C09083=1072.858,202.514,-79.918,173.836,27.136,154.832
C09084=1072.852,202.266,-79.894,173.834,27.133,154.832
C09085=1072.846,202.016,-79.870,173.831,27.130,154.831
C09086=1072.840,201.767,-79.847,173.830,27.128,154.831
C09087=1072.835,201.519,-79.822,173.827,27.125,154.831
C09088=1072.828,201.270,-79.798,173.825,27.122,154.830
C09089=1072.823,201.021,-79.774,173.822,27.119,154.830
C09090=1072.817,200.772,-79.751,173.820,27.116,154.830
C09091=1072.811,200.524,-79.727,173.819,27.114,154.829
C09092=1072.805,200.275,-79.703,173.816,27.110,154.829
C09093=1072.800,200.026,-79.680,173.814,27.107,154.828
C09094=1072.794,199.777,-79.656,173.811,27.104,154.828
C09095=1072.788,199.529,-79.632,173.810,27.102,154.828
C09096=1072.783,199.279,-79.608,173.807,27.099,154.827
C09097=1072.777,199.031,-79.584,173.805,27.096,154.827
C09098=1072.771,198.783,-79.561,173.802,27.093,154.827
C09099=1072.766,198.533,-79.537,173.801,27.090,154.826
C09100=1072.759,198.284,-79.513,173.799,27.087,154.826
C09101=1072.754,198.035,-79.490,173.796,27.085,154.826
C09102=1072.748,197.787,-79.466,173.794,27.082,154.825
C09103=1072.743,197.538,-79.442,173.792,27.079,154.825
C09104=1072.737,197.289,-79.419,173.790,27.076,154.824
C09105=1072.730,197.040,-79.395,173.787,27.073,154.824
C09106=1072.725,196.791,-79.371,173.785,27.070,154.824
C09107=1072.719,196.543,-79.348,173.783,27.068,154.823
C09108=1072.714,196.294,-79.325,173.781,27.065,154.823
C09109=1072.708,196.045,-79.300,173.779,27.062,154.823
C09110=1072.702,195.797,-79.277,173.776,27.059,154.822
C09111=1072.697,195.547,-79.253,173.775,27.056,154.822
C09112=1072.691,195.298,-79.230,173.772,27.053,154.821
C09113=1072.685,195.050,-79.206,173.770,27.050,154.821
C09114=1072.680,194.801,-79.183,173.768,27.047,154.821
C09115=1072.674,194.552,-79.160,173.766,27.044,154.820
C09116=1072.668,194.304,-79.136,173.764,27.041,154.820
C09117=1072.663,194.054,-79.112,173.761,27.039,154.820
C09118=1072.657,193.806,-79.089,173.760,27.036,154.819
C09119=1072.651,193.556,-79.065,173.757,27.033,154.819
C09120=1072.646,193.307,-79.042,173.755,27.030,154.818
C09121=1072.640,193.059,-79.018,173.753,27.027,154.818
C09122=1072.635,192.810,-78.995,173.751,27.025,154.818
C09123=1072.629,192.562,-78.971,173.748,27.022,154.817
C09124=1072.623,192.313,-78.948,173.747,27.019,154.817
C09125=1072.618,192.064,-78.925,173.745,27.016,154.817
C09126=1072.612,191.815,-78.901,173.742,27.013,154.816
C09127=1072.606,191.533,-78.875,173.740,27.010,154.816
C09128=1072.599,191.252,-78.848,173.737,27.007,154.815
C09129=1072.593,190.970,-78.822,173.735,27.003,154.815
C09130=1072.587,190.689,-78.796,173.733,27.000,154.815
C09131=1072.581,190.441,-78.772,173.730,26.997,154.814
C09132=1072.575,190.192,-78.749,173.729,26.994,154.814
C09133=1072.570,189.943,-78.726,173.726,26.991,154.813
C09134=1072.565,189.694,-78.703,173.724,26.989,154.813
C09135=1072.559,189.445,-78.679,173.722,26.986,154.813
C09136=1072.553,189.196,-78.656,173.720,26.983,154.812
C09137=1072.548,188.947,-78.633,173.718,26.980,154.812
C09138=1072.542,188.698,-78.610,173.716,26.977,154.811
C09139=1072.537,188.449,-78.587,173.714,26.974,154.811
C09140=1072.531,188.201,-78.563,173.711,26.972,154.811
C09141=1072.526,187.952,-78.539,173.710,26.969,154.810
C09142=1072.520,187.703,-78.517,173.707,26.966,154.810
C09143=1072.514,187.454,-78.494,173.705,26.963,154.810
C09144=1072.508,187.205,-78.471,173.704,26.960,154.809
C09145=1072.503,186.956,-78.447,173.701,26.957,154.809
C09146=1072.498,186.707,-78.424,173.700,26.955,154.809
C09147=1072.492,186.458,-78.401,173.697,26.952,154.808
C09148=1072.486,186.209,-78.378,173.695,26.949,154.808
C09149=1072.481,185.961,-78.354,173.693,26.946,154.807
C09150=1072.475,185.712,-78.331,173.691,26.943,154.807
C09151=1072.469,185.463,-78.308,173.689,26.940,154.807
C09152=1072.464,185.215,-78.286,173.687,26.937,154.806
C09153=1072.459,184.966,-78.262,173.685,26.934,154.806
C09154=1072.454,184.717,-78.239,173.682,26.931,154.806
C09155=1072.448,184.468,-78.216,173.681,26.929,154.805
C09156=1072.441,184.219,-78.194,173.678,26.926,154.805
C09157=1072.436,183.970,-78.171,173.677,26.923,154.804
C09158=1072.430,183.721,-78.148,173.674,26.921,154.804
C09159=1072.424,183.472,-78.126,173.672,26.918,154.804
C09160=1072.419,183.223,-78.103,173.671,26.915,154.803
C09161=1072.413,182.974,-78.080,173.668,26.912,154.803
C09162=1072.407,182.725,-78.057,173.666,26.909,154.803
C09163=1072.401,182.477,-78.034,173.664,26.907,154.802
C09164=1072.395,182.228,-78.012,173.662,26.904,154.802
C09165=1072.389,181.979,-77.989,173.660,26.901,154.802
C09166=1072.384,181.730,-77.966,173.658,26.899,154.801
C09167=1072.377,181.481,-77.943,173.655,26.896,154.801
C09168=1072.372,181.232,-77.921,173.654,26.893,154.801
C09169=1072.366,180.983,-77.898,173.651,26.890,154.800
C09170=1072.360,180.734,-77.875,173.650,26.888,154.800
C09171=1072.355,180.485,-77.852,173.647,26.885,154.800
C09172=1072.348,180.237,-77.830,173.645,26.882,154.799
C09173=1072.343,179.987,-77.808,173.644,26.880,154.799
C09174=1072.337,179.738,-77.785,173.641,26.877,154.799
C09175=1072.331,179.489,-77.762,173.640,26.874,154.798
C09176=1072.325,179.240,-77.739,173.637,26.871,154.798
C09177=1072.319,178.992,-77.716,173.635,26.868,154.798
C09178=1072.314,178.743,-77.695,173.633,26.866,154.797
C09179=1072.308,178.494,-77.672,173.631,26.863,154.797
C09180=1072.303,178.245,-77.649,173.629,26.860,154.796
C09181=1072.296,177.996,-77.627,173.627,26.858,154.796
C09182=1072.291,177.747,-77.604,173.625,26.855,154.796
C09183=1072.285,177.498,-77.581,173.623,26.852,154.795
C09184=1072.280,177.249,-77.559,173.621,26.849,154.795
C09185=1072.273,177.000,-77.537,173.619,26.847,154.795
C09186=1072.268,176.752,-77.514,173.617,26.844,154.794
C09187=1072.263,176.502,-77.492,173.615,26.841,154.794
C09188=1072.257,176.253,-77.469,173.613,26.838,154.794
C09189=1072.250,176.005,-77.446,173.610,26.836,154.793
C09190=1072.245,175.755,-77.424,173.609,26.833,154.793
C09191=1072.239,175.475,-77.399,173.607,26.830,154.793
C09192=1072.233,175.192,-77.373,173.604,26.827,154.792
C09193=1072.226,174.910,-77.348,173.602,26.824,154.792
C09194=1072.219,174.629,-77.322,173.599,26.821,154.792
C09195=1072.213,174.379,-77.300,173.598,26.818,154.791
C09196=1072.208,174.131,-77.277,173.596,26.815,154.791
C09197=1072.202,173.882,-77.256,173.594,26.813,154.790
C09198=1072.196,173.633,-77.233,173.592,26.810,154.790
C09199=1072.191,173.383,-77.211,173.590,26.807,154.790
C09200=1072.185,173.135,-77.189,173.588,26.804,154.789
C09201=1072.180,172.886,-77.166,173.586,26.802,154.789
C09202=1072.174,172.637,-77.144,173.584,26.798,154.789
C09203=1072.168,172.388,-77.122,173.581,26.796,154.788
C09204=1072.163,172.140,-77.099,173.580,26.793,154.788
C09205=1072.157,171.890,-77.077,173.578,26.790,154.788
C09206=1072.151,171.641,-77.055,173.576,26.788,154.787
C09207=1072.145,171.392,-77.032,173.574,26.785,154.787
C09208=1072.140,171.143,-77.011,173.572,26.782,154.786
C09209=1072.134,170.895,-76.988,173.570,26.779,154.786
C09210=1072.129,170.645,-76.966,173.568,26.777,154.786
C09211=1072.123,170.397,-76.943,173.566,26.774,154.785
C09212=1072.117,170.148,-76.922,173.564,26.771,154.785
C09213=1072.112,169.898,-76.900,173.562,26.768,154.785
C09214=1072.107,169.650,-76.877,173.561,26.765,154.784
C09215=1072.101,169.401,-76.855,173.558,26.762,154.784
C09216=1072.095,169.152,-76.832,173.557,26.760,154.784
C09217=1072.089,168.902,-76.810,173.554,26.757,154.783
C09218=1072.084,168.654,-76.789,173.553,26.754,154.783
C09219=1072.078,168.405,-76.766,173.550,26.752,154.783
C09220=1072.073,168.156,-76.744,173.549,26.749,154.782
C09221=1072.067,167.907,-76.722,173.546,26.746,154.782
C09222=1072.062,167.657,-76.700,173.545,26.744,154.781
C09223=1072.056,167.410,-76.678,173.543,26.741,154.781
C09224=1072.050,167.160,-76.656,173.541,26.738,154.781
C09225=1072.045,166.910,-76.634,173.539,26.735,154.780
C09226=1072.039,166.663,-76.612,173.537,26.733,154.780
C09227=1072.034,166.413,-76.590,173.535,26.729,154.780
C09228=1072.028,166.165,-76.568,173.533,26.727,154.779
C09229=1072.023,165.915,-76.546,173.531,26.724,154.779
C09230=1072.017,165.666,-76.524,173.529,26.721,154.779
C09231=1072.011,165.418,-76.502,173.527,26.718,154.778
C09232=1072.006,165.168,-76.480,173.526,26.715,154.778
C09233=1072.000,164.920,-76.458,173.523,26.713,154.778
C09234=1071.995,164.670,-76.436,173.522,26.710,154.777
C09235=1071.990,164.421,-76.414,173.519,26.707,154.777
C09236=1071.984,164.173,-76.392,173.518,26.704,154.776
C09237=1071.978,163.923,-76.370,173.516,26.702,154.776
C09238=1071.973,163.675,-76.348,173.514,26.699,154.776
C09239=1071.967,163.425,-76.326,173.513,26.696,154.775
C09240=1071.962,163.177,-76.305,173.510,26.693,154.775
C09241=1071.956,162.927,-76.283,173.509,26.691,154.775
C09242=1071.951,162.679,-76.261,173.506,26.688,154.774
C09243=1071.945,162.429,-76.239,173.505,26.685,154.774
C09244=1071.940,162.180,-76.217,173.503,26.682,154.773
C09245=1071.934,161.931,-76.196,173.501,26.680,154.773
C09246=1071.929,161.683,-76.173,173.499,26.677,154.773
C09247=1071.923,161.434,-76.151,173.497,26.674,154.772
C09248=1071.918,161.185,-76.130,173.496,26.671,154.772
C09249=1071.912,160.936,-76.108,173.493,26.668,154.772
C09250=1071.906,160.687,-76.087,173.492,26.666,154.771
C09251=1071.900,160.438,-76.065,173.489,26.663,154.771
C09252=1071.895,160.188,-76.043,173.488,26.660,154.771
C09253=1071.889,159.940,-76.022,173.486,26.657,154.770
C09254=1071.883,159.690,-76.001,173.484,26.655,154.770
C09255=1071.877,159.409,-75.976,173.482,26.652,154.770
C09256=1071.871,159.126,-75.952,173.479,26.649,154.769
C09257=1071.864,158.844,-75.927,173.478,26.646,154.769
C09258=1071.858,158.561,-75.902,173.476,26.643,154.768
C09259=1071.852,158.313,-75.881,173.473,26.640,154.768
C09260=1071.846,158.064,-75.859,173.472,26.637,154.768
C09261=1071.840,157.815,-75.838,173.469,26.634,154.767
C09262=1071.834,157.566,-75.816,173.468,26.632,154.767
C09263=1071.830,157.316,-75.795,173.466,26.629,154.767
C09264=1071.824,157.067,-75.774,173.464,26.626,154.766
C09265=1071.818,156.819,-75.752,173.463,26.624,154.766
C09266=1071.812,156.569,-75.731,173.460,26.621,154.766
C09267=1071.806,156.321,-75.709,173.459,26.618,154.765
C09268=1071.801,156.071,-75.687,173.456,26.615,154.765
C09269=1071.796,155.822,-75.667,173.455,26.613,154.764
C09270=1071.789,155.573,-75.645,173.453,26.610,154.764
C09271=1071.784,155.325,-75.624,173.451,26.608,154.764
C09272=1071.778,155.075,-75.602,173.449,26.605,154.763
C09273=1071.772,154.827,-75.581,173.447,26.602,154.763
C09274=1071.766,154.577,-75.560,173.446,26.599,154.763
C09275=1071.761,154.329,-75.539,173.444,26.597,154.762
C09276=1071.755,154.079,-75.516,173.442,26.594,154.762
C09277=1071.750,153.831,-75.495,173.440,26.591,154.762
C09278=1071.745,153.581,-75.475,173.438,26.589,154.761
C09279=1071.738,153.332,-75.453,173.436,26.586,154.761
C09280=1071.733,153.084,-75.432,173.435,26.583,154.761
C09281=1071.727,152.834,-75.411,173.432,26.581,154.760
C09282=1071.721,152.585,-75.390,173.431,26.578,154.760
C09283=1071.715,152.336,-75.368,173.429,26.575,154.760
C09284=1071.710,152.087,-75.347,173.427,26.572,154.759
C09285=1071.704,151.838,-75.326,173.426,26.570,154.759
C09286=1071.698,151.589,-75.304,173.423,26.567,154.759
C09287=1071.693,151.340,-75.284,173.422,26.564,154.758
C09288=1071.687,151.091,-75.262,173.419,26.561,154.758
C09289=1071.681,150.843,-75.241,173.418,26.559,154.757
C09290=1071.675,150.593,-75.220,173.417,26.556,154.757
C09291=1071.670,150.344,-75.199,173.414,26.554,154.757
C09292=1071.665,150.095,-75.178,173.413,26.551,154.756
C09293=1071.658,149.846,-75.157,173.411,26.548,154.756
C09294=1071.653,149.597,-75.135,173.409,26.545,154.756
C09295=1071.647,149.348,-75.114,173.407,26.543,154.755
C09296=1071.641,149.099,-75.093,173.405,26.540,154.755
C09297=1071.636,148.850,-75.073,173.403,26.537,154.755
C09298=1071.630,148.601,-75.051,173.402,26.534,154.754
C09299=1071.625,148.352,-75.030,173.400,26.532,154.754
C09300=1071.619,148.102,-75.009,173.398,26.529,154.754
C09301=1071.613,147.853,-74.988,173.397,26.527,154.753
C09302=1071.608,147.605,-74.967,173.394,26.524,154.753
C09303=1071.602,147.355,-74.946,173.393,26.521,154.753
C09304=1071.596,147.107,-74.925,173.390,26.518,154.752
C09305=1071.590,146.858,-74.905,173.389,26.516,154.752
C09306=1071.584,146.608,-74.883,173.387,26.513,154.752
C09307=1071.579,146.359,-74.863,173.385,26.510,154.751
C09308=1071.573,146.109,-74.842,173.384,26.508,154.751
C09309=1071.567,145.861,-74.821,173.382,26.505,154.750
C09310=1071.562,145.612,-74.800,173.380,26.502,154.750
C09311=1071.555,145.363,-74.779,173.378,26.500,154.750
C09312=1071.550,145.114,-74.758,173.377,26.497,154.749
C09313=1071.545,144.865,-74.738,173.374,26.494,154.749
C09314=1071.539,144.615,-74.716,173.373,26.492,154.749
C09315=1071.533,144.367,-74.696,173.371,26.489,154.748
C09316=1071.527,144.118,-74.676,173.369,26.486,154.748
C09317=1071.521,143.868,-74.654,173.368,26.484,154.748
C09318=1071.516,143.619,-74.633,173.366,26.481,154.747
C09319=1071.509,143.337,-74.610,173.364,26.478,154.747
C09320=1071.503,143.054,-74.586,173.361,26.475,154.747
C09321=1071.496,142.772,-74.563,173.360,26.472,154.746
C09322=1071.490,142.489,-74.540,173.358,26.469,154.746
C09323=1071.484,142.241,-74.519,173.356,26.466,154.745
C09324=1071.479,141.991,-74.498,173.354,26.463,154.745
C09325=1071.473,141.742,-74.477,173.352,26.461,154.745
C09326=1071.467,141.494,-74.456,173.351,26.458,154.744
C09327=1071.461,141.244,-74.436,173.349,26.455,154.744
C09328=1071.456,140.995,-74.415,173.347,26.453,154.744
C09329=1071.451,140.746,-74.394,173.346,26.450,154.743
C09330=1071.444,140.498,-74.374,173.343,26.447,154.743
C09331=1071.438,140.248,-74.353,173.342,26.445,154.743
C09332=1071.433,139.999,-74.332,173.340,26.442,154.742
C09333=1071.427,139.750,-74.312,173.338,26.439,154.742
C09334=1071.422,139.501,-74.292,173.337,26.436,154.742
C09335=1071.416,139.251,-74.271,173.335,26.434,154.741
C09336=1071.410,139.003,-74.250,173.333,26.431,154.741
C09337=1071.405,138.754,-74.230,173.331,26.428,154.740
C09338=1071.399,138.504,-74.209,173.330,26.426,154.740
C09339=1071.393,138.255,-74.189,173.327,26.423,154.740
C09340=1071.387,138.006,-74.168,173.326,26.421,154.740
C09341=1071.381,137.757,-74.148,173.325,26.418,154.739
C09342=1071.376,137.508,-74.128,173.323,26.415,154.739
C09343=1071.370,137.258,-74.107,173.321,26.412,154.738
C09344=1071.364,137.010,-74.086,173.319,26.410,154.738
C09345=1071.359,136.761,-74.066,173.318,26.407,154.738
C09346=1071.353,136.512,-74.046,173.315,26.404,154.737
C09347=1071.348,136.263,-74.025,173.314,26.402,154.737
C09348=1071.341,136.013,-74.005,173.312,26.399,154.737
C09349=1071.336,135.764,-73.984,173.310,26.396,154.736
C09350=1071.330,135.515,-73.964,173.309,26.394,154.736
C09351=1071.324,135.266,-73.944,173.307,26.391,154.736
C09352=1071.318,135.017,-73.924,173.306,26.389,154.735
C09353=1071.313,134.768,-73.903,173.303,26.386,154.735
C09354=1071.307,134.519,-73.883,173.302,26.383,154.735
C09355=1071.301,134.270,-73.862,173.300,26.380,154.734
C09356=1071.295,134.021,-73.842,173.298,26.377,154.734
C09357=1071.290,133.772,-73.822,173.297,26.375,154.734
C09358=1071.285,133.523,-73.801,173.295,26.372,154.733
C09359=1071.278,133.273,-73.781,173.293,26.369,154.733
C09360=1071.273,133.024,-73.760,173.291,26.367,154.733
C09361=1071.267,132.775,-73.740,173.290,26.364,154.732
C09362=1071.262,132.525,-73.721,173.289,26.361,154.732
C09363=1071.256,132.277,-73.701,173.286,26.359,154.731
C09364=1071.251,132.027,-73.680,173.285,26.356,154.731
C09365=1071.245,131.779,-73.660,173.283,26.354,154.731
C09366=1071.238,131.529,-73.640,173.282,26.351,154.730
C09367=1071.232,131.280,-73.620,173.279,26.348,154.730
C09368=1071.227,131.031,-73.599,173.278,26.345,154.730
C09369=1071.221,130.782,-73.579,173.276,26.343,154.729
C09370=1071.215,130.533,-73.560,173.274,26.340,154.729
C09371=1071.209,130.283,-73.539,173.273,26.338,154.729
C09372=1071.203,130.034,-73.519,173.271,26.335,154.728
C09373=1071.197,129.785,-73.499,173.270,26.333,154.728
C09374=1071.191,129.537,-73.479,173.267,26.330,154.728
C09375=1071.186,129.287,-73.459,173.266,26.327,154.727
C09376=1071.180,129.038,-73.439,173.264,26.324,154.727
C09377=1071.174,128.789,-73.419,173.263,26.322,154.727
C09378=1071.168,128.540,-73.399,173.261,26.319,154.726
C09379=1071.163,128.291,-73.379,173.259,26.316,154.726
C09380=1071.157,128.041,-73.359,173.258,26.314,154.726
C09381=1071.151,127.792,-73.339,173.255,26.311,154.725
C09382=1071.145,127.544,-73.319,173.254,26.309,154.725
C09383=1071.138,127.261,-73.296,173.252,26.306,154.725
C09384=1071.132,126.978,-73.274,173.250,26.303,154.724
C09385=1071.126,126.695,-73.252,173.249,26.300,154.724
C09386=1071.118,126.413,-73.229,173.246,26.297,154.723
C09387=1071.113,126.163,-73.209,173.245,26.294,154.723
C09388=1071.107,125.915,-73.189,173.244,26.291,154.723
C09389=1071.101,125.665,-73.170,173.241,26.288,154.722
C09390=1071.095,125.416,-73.150,173.240,26.286,154.722
C09391=1071.090,125.167,-73.130,173.238,26.283,154.722
C09392=1071.084,124.918,-73.110,173.237,26.281,154.721
C09393=1071.078,124.669,-73.090,173.234,26.277,154.721
C09394=1071.073,124.420,-73.071,173.233,26.275,154.721
C09395=1071.067,124.171,-73.051,173.232,26.272,154.720
C09396=1071.061,123.922,-73.030,173.230,26.270,154.720
C09397=1071.056,123.672,-73.011,173.228,26.267,154.720
C09398=1071.050,123.423,-72.991,173.226,26.264,154.719
C09399=1071.044,123.174,-72.972,173.225,26.262,154.719
C09400=1071.038,122.925,-72.952,173.223,26.259,154.718
C09401=1071.032,122.676,-72.932,173.221,26.256,154.718
C09402=1071.027,122.427,-72.912,173.220,26.254,154.718
C09403=1071.021,122.178,-72.892,173.218,26.251,154.717
C09404=1071.015,121.928,-72.873,173.217,26.249,154.717
C09405=1071.009,121.680,-72.853,173.214,26.245,154.717
C09406=1071.004,121.430,-72.833,173.213,26.243,154.716
C09407=1070.998,121.181,-72.813,173.211,26.240,154.716
C09408=1070.993,120.932,-72.794,173.210,26.237,154.716
C09409=1070.987,120.683,-72.774,173.209,26.235,154.715
C09410=1070.981,120.433,-72.754,173.206,26.232,154.715
C09411=1070.975,120.185,-72.734,173.205,26.229,154.715
C09412=1070.969,119.935,-72.715,173.203,26.227,154.714
C09413=1070.964,119.686,-72.696,173.202,26.224,154.714
C09414=1070.958,119.437,-72.676,173.200,26.221,154.713
C09415=1070.953,119.187,-72.656,173.198,26.219,154.713
C09416=1070.947,118.938,-72.636,173.197,26.216,154.713
C09417=1070.941,118.689,-72.617,173.195,26.213,154.712
C09418=1070.935,118.440,-72.597,173.194,26.211,154.712
C09419=1070.929,118.191,-72.578,173.192,26.208,154.712
C09420=1070.924,117.941,-72.559,173.190,26.205,154.711
C09421=1070.918,117.692,-72.539,173.189,26.203,154.711
C09422=1070.912,117.443,-72.519,173.187,26.200,154.711
C09423=1070.908,117.194,-72.500,173.186,26.197,154.710
C09424=1070.902,116.945,-72.480,173.183,26.194,154.710
C09425=1070.896,116.696,-72.461,173.182,26.191,154.710
C09426=1070.890,116.447,-72.441,173.181,26.189,154.709
C09427=1070.884,116.197,-72.421,173.179,26.186,154.709
C09428=1070.879,115.948,-72.402,173.178,26.184,154.708
C09429=1070.873,115.699,-72.383,173.175,26.180,154.708
C09430=1070.867,115.450,-72.363,173.174,26.178,154.708
C09431=1070.862,115.201,-72.344,173.173,26.175,154.707
C09432=1070.856,114.952,-72.325,173.171,26.172,154.707
C09433=1070.851,114.702,-72.304,173.170,26.170,154.707
C09434=1070.845,114.453,-72.285,173.167,26.166,154.706
C09435=1070.840,114.204,-72.266,173.166,26.164,154.706
C09436=1070.833,113.954,-72.247,173.165,26.161,154.705
C09437=1070.827,113.706,-72.227,173.163,26.159,154.705
C09438=1070.822,113.456,-72.208,173.162,26.156,154.705
C09439=1070.816,113.207,-72.189,173.159,26.153,154.704
C09440=1070.811,112.958,-72.170,173.158,26.151,154.704
C09441=1070.805,112.709,-72.151,173.157,26.148,154.704
C09442=1070.799,112.460,-72.131,173.155,26.145,154.703
C09443=1070.793,112.210,-72.111,173.154,26.143,154.703
C09444=1070.788,111.961,-72.092,173.152,26.140,154.703
C09445=1070.781,111.712,-72.074,173.150,26.137,154.702
C09446=1070.776,111.462,-72.054,173.148,26.135,154.702
C09447=1070.769,111.180,-72.032,173.147,26.132,154.702
C09448=1070.763,110.897,-72.010,173.145,26.129,154.701
C09449=1070.756,110.615,-71.989,173.143,26.126,154.701
C09450=1070.749,110.332,-71.968,173.141,26.123,154.700
C09451=1070.744,110.083,-71.948,173.140,26.120,154.700
C09452=1070.738,109.833,-71.929,173.138,26.117,154.700
C09453=1070.732,109.584,-71.910,173.137,26.115,154.699
C09454=1070.726,109.336,-71.891,173.135,26.112,154.699
C09455=1070.720,109.087,-71.872,173.133,26.109,154.699
C09456=1070.715,108.837,-71.852,173.132,26.106,154.698
C09457=1070.709,108.588,-71.833,173.130,26.104,154.698
C09458=1070.703,108.339,-71.814,173.129,26.101,154.698
C09459=1070.697,108.089,-71.795,173.127,26.098,154.697
C09460=1070.692,107.840,-71.776,173.125,26.096,154.697
C09461=1070.685,107.591,-71.758,173.124,26.093,154.697
C09462=1070.680,107.342,-71.738,173.122,26.090,154.696
C09463=1070.674,107.092,-71.719,173.121,26.088,154.696
C09464=1070.668,106.843,-71.700,173.119,26.085,154.695
C09465=1070.662,106.595,-71.682,173.118,26.082,154.695
C09466=1070.657,106.345,-71.662,173.115,26.080,154.695
C09467=1070.651,106.096,-71.643,173.114,26.077,154.694
C09468=1070.645,105.847,-71.625,173.113,26.074,154.694
C09469=1070.639,105.597,-71.605,173.111,26.072,154.694
C09470=1070.634,105.348,-71.586,173.110,26.069,154.693
C09471=1070.627,105.099,-71.568,173.108,26.067,154.693
C09472=1070.622,104.849,-71.549,173.107,26.064,154.693
C09473=1070.616,104.600,-71.530,173.105,26.061,154.692
C09474=1070.611,104.351,-71.512,173.103,26.058,154.692
C09475=1070.605,104.102,-71.492,173.102,26.055,154.692
C09476=1070.599,103.853,-71.473,173.100,26.053,154.691
C09477=1070.593,103.603,-71.455,173.099,26.050,154.691
C09478=1070.588,103.355,-71.436,173.098,26.047,154.690
C09479=1070.582,103.105,-71.416,173.095,26.044,154.690
C09480=1070.576,102.856,-71.398,173.094,26.041,154.690
C09481=1070.570,102.606,-71.379,173.092,26.039,154.689
C09482=1070.565,102.357,-71.360,173.091,26.036,154.689
C09483=1070.559,102.108,-71.342,173.090,26.033,154.689
C09484=1070.553,101.859,-71.323,173.088,26.031,154.688
C09485=1070.548,101.610,-71.304,173.087,26.028,154.688
C09486=1070.541,101.361,-71.285,173.085,26.025,154.687
C09487=1070.536,101.111,-71.266,173.083,26.023,154.687
C09488=1070.530,100.862,-71.248,173.082,26.020,154.687
C09489=1070.525,100.613,-71.229,173.080,26.017,154.686
C09490=1070.518,100.364,-71.210,173.079,26.015,154.686
C09491=1070.513,100.114,-71.192,173.077,26.012,154.686
C09492=1070.506,99.865,-71.173,173.076,26.010,154.685
C09493=1070.501,99.616,-71.154,173.074,26.007,154.685
C09494=1070.495,99.367,-71.136,173.072,26.004,154.685
C09495=1070.489,99.117,-71.117,173.071,26.001,154.684
C09496=1070.484,98.868,-71.099,173.069,25.999,154.684
C09497=1070.478,98.619,-71.080,173.068,25.996,154.684
C09498=1070.472,98.369,-71.062,173.067,25.994,154.683
C09499=1070.465,98.120,-71.043,173.065,25.991,154.683
C09500=1070.460,97.871,-71.024,173.063,25.988,154.683
C09501=1070.454,97.622,-71.006,173.061,25.985,154.682
C09502=1070.449,97.372,-70.987,173.060,25.982,154.682
C09503=1070.443,97.124,-70.969,173.059,25.980,154.682
C09504=1070.437,96.874,-70.950,173.057,25.977,154.681
C09505=1070.431,96.625,-70.931,173.056,25.975,154.681
C09506=1070.425,96.376,-70.913,173.054,25.972,154.680
C09507=1070.420,96.126,-70.895,173.053,25.969,154.680
C09508=1070.413,95.877,-70.876,173.051,25.967,154.680
C09509=1070.408,95.628,-70.857,173.049,25.964,154.679
C09510=1070.402,95.379,-70.839,173.048,25.961,154.679
C09511=1070.395,95.096,-70.818,173.046,25.958,154.679
C09512=1070.390,94.813,-70.798,173.044,25.955,154.678
C09513=1070.382,94.531,-70.777,173.043,25.952,154.678
C09514=1070.375,94.248,-70.755,173.040,25.949,154.677
C09515=1070.370,93.998,-70.737,173.039,25.946,154.677
C09516=1070.364,93.750,-70.719,173.038,25.943,154.677
C09517=1070.358,93.500,-70.701,173.036,25.941,154.676
C09518=1070.353,93.252,-70.682,173.035,25.938,154.676
C09519=1070.347,93.002,-70.664,173.034,25.935,154.676
C09520=1070.341,92.752,-70.645,173.032,25.933,154.675
C09521=1070.336,92.503,-70.627,173.031,25.930,154.675
C09522=1070.329,92.254,-70.608,173.029,25.927,154.674
C09523=1070.325,92.005,-70.590,173.027,25.924,154.674
C09524=1070.318,91.756,-70.572,173.026,25.922,154.674
C09525=1070.313,91.507,-70.554,173.024,25.919,154.673
C09526=1070.307,91.257,-70.535,173.023,25.916,154.673
C09527=1070.301,91.008,-70.517,173.021,25.914,154.673
C09528=1070.295,90.759,-70.499,173.020,25.911,154.672
C09529=1070.290,90.509,-70.480,173.019,25.908,154.672
C09530=1070.284,90.260,-70.462,173.017,25.906,154.672
C09531=1070.278,90.011,-70.444,173.016,25.903,154.671
C09532=1070.271,89.761,-70.426,173.013,25.900,154.671
C09533=1070.266,89.513,-70.408,173.012,25.897,154.671
C09534=1070.260,89.263,-70.390,173.011,25.895,154.670
C09535=1070.254,89.014,-70.372,173.009,25.892,154.670
C09536=1070.248,88.765,-70.353,173.008,25.889,154.669
C09537=1070.242,88.515,-70.335,173.006,25.887,154.669
C09538=1070.237,88.266,-70.317,173.005,25.884,154.669
C09539=1070.230,88.017,-70.299,173.004,25.881,154.668
C09540=1070.225,87.768,-70.281,173.002,25.879,154.668
C09541=1070.219,87.518,-70.263,173.000,25.876,154.668
C09542=1070.213,87.269,-70.245,172.998,25.873,154.667
C09543=1070.207,87.019,-70.226,172.997,25.871,154.667
C09544=1070.201,86.770,-70.208,172.996,25.868,154.667
C09545=1070.195,86.521,-70.190,172.994,25.865,154.666
C09546=1070.189,86.271,-70.172,172.993,25.863,154.666
C09547=1070.184,86.022,-70.155,172.991,25.860,154.666
C09548=1070.178,85.773,-70.137,172.990,25.858,154.665
C09549=1070.172,85.524,-70.118,172.989,25.855,154.665
C09550=1070.166,85.275,-70.101,172.987,25.852,154.664
C09551=1070.160,85.025,-70.083,172.985,25.849,154.664
C09552=1070.155,84.775,-70.064,172.983,25.846,154.664
C09553=1070.149,84.527,-70.046,172.982,25.844,154.663
C09554=1070.143,84.277,-70.028,172.981,25.841,154.663
C09555=1070.137,84.028,-70.011,172.979,25.838,154.663
C09556=1070.131,83.778,-69.993,172.978,25.836,154.662
C09557=1070.126,83.529,-69.975,172.976,25.833,154.662
C09558=1070.119,83.280,-69.956,172.975,25.830,154.662
C09559=1070.114,83.031,-69.939,172.974,25.828,154.661
C09560=1070.108,82.782,-69.921,172.972,25.825,154.661
C09561=1070.102,82.532,-69.903,172.970,25.822,154.661
C09562=1070.096,82.283,-69.885,172.969,25.819,154.660
C09563=1070.091,82.034,-69.868,172.967,25.816,154.660
C09564=1070.084,81.785,-69.849,172.966,25.814,154.659
C09565=1070.079,81.535,-69.831,172.964,25.811,154.659
C09566=1070.074,81.286,-69.814,172.963,25.808,154.659
C09567=1070.068,81.036,-69.796,172.962,25.806,154.658
C09568=1070.062,80.787,-69.778,172.960,25.803,154.658
C09569=1070.056,80.538,-69.760,172.959,25.800,154.658
C09570=1070.051,80.289,-69.743,172.957,25.798,154.657
C09571=1070.044,80.039,-69.725,172.956,25.795,154.657
C09572=1070.039,79.790,-69.707,172.955,25.792,154.656
C09573=1070.033,79.541,-69.689,172.952,25.789,154.656
C09574=1070.027,79.292,-69.671,172.951,25.787,154.656
C09575=1070.020,79.009,-69.651,172.950,25.783,154.655
C09576=1070.014,78.726,-69.630,172.948,25.780,154.655
C09577=1070.008,78.444,-69.611,172.946,25.777,154.655
C09578=1070.000,78.161,-69.591,172.945,25.774,154.654
C09579=1069.995,77.912,-69.573,172.943,25.772,154.654
C09580=1069.989,77.663,-69.556,172.942,25.769,154.653
C09581=1069.983,77.413,-69.538,172.941,25.766,154.653
C09582=1069.978,77.164,-69.520,172.939,25.764,154.653
C09583=1069.971,76.915,-69.503,172.938,25.761,154.652
C09584=1069.965,76.666,-69.485,172.936,25.758,154.652
C09585=1069.959,76.416,-69.467,172.934,25.755,154.652
C09586=1069.954,76.167,-69.450,172.933,25.753,154.651
C09587=1069.948,75.918,-69.432,172.931,25.750,154.651
C09588=1069.942,75.668,-69.415,172.930,25.748,154.651
C09589=1069.936,75.419,-69.398,172.929,25.745,154.650
C09590=1069.930,75.169,-69.380,172.927,25.742,154.650
C09591=1069.925,74.920,-69.362,172.926,25.740,154.650
C09592=1069.919,74.671,-69.345,172.924,25.737,154.649
C09593=1069.913,74.421,-69.327,172.923,25.734,154.649
C09594=1069.907,74.172,-69.309,172.922,25.732,154.648
C09595=1069.901,73.923,-69.292,172.920,25.729,154.648
C09596=1069.895,73.674,-69.274,172.919,25.726,154.648
C09597=1069.890,73.424,-69.258,172.917,25.723,154.647
C09598=1069.884,73.174,-69.240,172.915,25.720,154.647
C09599=1069.878,72.925,-69.222,172.914,25.718,154.647
C09600=1069.872,72.677,-69.205,172.912,25.715,154.646
C09601=1069.866,72.427,-69.187,172.911,25.712,154.646
C09602=1069.860,72.178,-69.170,172.910,25.709,154.645
C09603=1069.855,71.928,-69.153,172.908,25.707,154.645
C09604=1069.848,71.679,-69.135,172.907,25.704,154.645
C09605=1069.843,71.430,-69.118,172.906,25.701,154.644
C09606=1069.837,71.181,-69.100,172.904,25.699,154.644
C09607=1069.831,70.931,-69.082,172.903,25.696,154.644
C09608=1069.825,70.682,-69.066,172.901,25.693,154.643
C09609=1069.820,70.432,-69.049,172.900,25.691,154.643
C09610=1069.813,70.183,-69.031,172.899,25.688,154.643
C09611=1069.808,69.934,-69.013,172.897,25.685,154.642
C09612=1069.802,69.684,-68.997,172.895,25.682,154.642
C09613=1069.796,69.435,-68.979,172.893,25.680,154.642
C09614=1069.790,69.186,-68.961,172.892,25.677,154.641
C09615=1069.784,68.936,-68.945,172.891,25.675,154.641
C09616=1069.779,68.687,-68.928,172.889,25.672,154.640
C09617=1069.772,68.438,-68.910,172.888,25.669,154.640
C09618=1069.767,68.188,-68.893,172.887,25.667,154.640
C09619=1069.761,67.939,-68.876,172.885,25.664,154.639
C09620=1069.754,67.690,-68.858,172.884,25.661,154.639
C09621=1069.749,67.440,-68.842,172.882,25.659,154.639
C09622=1069.744,67.191,-68.824,172.881,25.656,154.638
C09623=1069.737,66.942,-68.807,172.880,25.653,154.638
C09624=1069.732,66.692,-68.790,172.878,25.650,154.638
C09625=1069.725,66.443,-68.773,172.877,25.648,154.637
C09626=1069.720,66.194,-68.755,172.876,25.645,154.637
C09627=1069.714,65.944,-68.738,172.874,25.642,154.637
C09628=1069.708,65.695,-68.721,172.873,25.640,154.636
C09629=1069.703,65.445,-68.704,172.871,25.636,154.636
C09630=1069.696,65.197,-68.687,172.869,25.634,154.635
C09631=1069.690,64.947,-68.669,172.868,25.631,154.635
C09632=1069.684,64.698,-68.653,172.866,25.628,154.635
C09633=1069.679,64.448,-68.635,172.865,25.626,154.634
C09634=1069.673,64.199,-68.619,172.864,25.623,154.634
C09635=1069.667,63.949,-68.601,172.862,25.621,154.634
C09636=1069.661,63.700,-68.585,172.861,25.618,154.633
C09637=1069.654,63.451,-68.568,172.859,25.616,154.633
C09638=1069.649,63.201,-68.551,172.858,25.613,154.633
C09639=1069.641,62.919,-68.532,172.857,25.610,154.632
C09640=1069.635,62.636,-68.513,172.854,25.607,154.632
C09641=1069.628,62.353,-68.493,172.853,25.604,154.631
C09642=1069.621,62.071,-68.474,172.852,25.601,154.631
C09643=1069.616,61.821,-68.458,172.850,25.598,154.631
C09644=1069.609,61.572,-68.440,172.849,25.596,154.630
C09645=1069.603,61.322,-68.424,172.847,25.592,154.630
C09646=1069.597,61.073,-68.406,172.845,25.590,154.630
C09647=1069.592,60.824,-68.390,172.844,25.587,154.629
C09648=1069.585,60.574,-68.373,172.842,25.585,154.629
C09649=1069.579,60.325,-68.356,172.841,25.582,154.629
C09650=1069.573,60.076,-68.339,172.840,25.579,154.628
C09651=1069.567,59.827,-68.323,172.838,25.577,154.628
C09652=1069.562,59.577,-68.306,172.837,25.574,154.628
C09653=1069.555,59.328,-68.288,172.836,25.572,154.627
C09654=1069.549,59.078,-68.272,172.834,25.569,154.627
C09655=1069.544,58.829,-68.255,172.833,25.566,154.626
C09656=1069.538,58.580,-68.238,172.831,25.564,154.626
C09657=1069.532,58.331,-68.222,172.830,25.561,154.626
C09658=1069.526,58.081,-68.204,172.829,25.558,154.626
C09659=1069.520,57.831,-68.188,172.827,25.556,154.625
C09660=1069.514,57.582,-68.172,172.826,25.553,154.625
C09661=1069.508,57.333,-68.155,172.825,25.550,154.624
C09662=1069.502,57.084,-68.138,172.823,25.547,154.624
C09663=1069.496,56.834,-68.121,172.822,25.545,154.624
C09664=1069.490,56.584,-68.105,172.820,25.542,154.623
C09665=1069.484,56.335,-68.087,172.819,25.539,154.623
C09666=1069.478,56.086,-68.071,172.817,25.537,154.623
C09667=1069.472,55.837,-68.055,172.815,25.534,154.622
C09668=1069.467,55.588,-68.037,172.814,25.532,154.622
C09669=1069.460,55.337,-68.021,172.813,25.529,154.622
C09670=1069.454,55.088,-68.004,172.811,25.526,154.621
C09671=1069.448,54.839,-67.988,172.810,25.523,154.621
C09672=1069.443,54.590,-67.971,172.808,25.521,154.621
C09673=1069.437,54.340,-67.954,172.807,25.518,154.620
C09674=1069.431,54.091,-67.938,172.806,25.515,154.620
C09675=1069.425,53.842,-67.922,172.804,25.512,154.619
C09676=1069.420,53.592,-67.905,172.803,25.510,154.619
C09677=1069.414,53.343,-67.888,172.802,25.507,154.619
C09678=1069.407,53.093,-67.871,172.800,25.504,154.618
C09679=1069.401,52.844,-67.855,172.799,25.502,154.618
C09680=1069.396,52.594,-67.838,172.797,25.499,154.618
C09681=1069.390,52.345,-67.822,172.796,25.496,154.617
C09682=1069.384,52.096,-67.806,172.795,25.494,154.617
C09683=1069.378,51.847,-67.789,172.793,25.491,154.617
C09684=1069.372,51.597,-67.772,172.792,25.488,154.616
C09685=1069.367,51.348,-67.756,172.791,25.486,154.616
C09686=1069.361,51.098,-67.739,172.789,25.483,154.616
C09687=1069.355,50.849,-67.723,172.788,25.481,154.615
C09688=1069.349,50.599,-67.706,172.787,25.478,154.615
C09689=1069.343,50.350,-67.690,172.785,25.475,154.614
C09690=1069.338,50.101,-67.674,172.784,25.473,154.614
C09691=1069.331,49.852,-67.657,172.782,25.469,154.614
C09692=1069.325,49.603,-67.641,172.780,25.466,154.613
C09693=1069.320,49.352,-67.623,172.779,25.464,154.613
C09694=1069.314,49.103,-67.607,172.777,25.461,154.613
C09695=1069.308,48.854,-67.591,172.776,25.458,154.612
C09696=1069.302,48.604,-67.575,172.775,25.456,154.612
C09697=1069.296,48.355,-67.558,172.773,25.453,154.612
C09698=1069.290,48.105,-67.542,172.772,25.450,154.611
C09699=1069.285,47.856,-67.525,172.771,25.448,154.611
C09700=1069.279,47.607,-67.509,172.769,25.445,154.611
C09701=1069.273,47.357,-67.493,172.768,25.442,154.610
C09702=1069.267,47.108,-67.477,172.766,25.440,154.610
C09703=1069.260,46.825,-67.458,172.765,25.436,154.609
C09704=1069.254,46.542,-67.440,172.764,25.433,154.609
C09705=1069.248,46.259,-67.421,172.762,25.430,154.609
C09706=1069.241,45.976,-67.403,172.760,25.427,154.608
C09707=1069.235,45.727,-67.386,172.759,25.424,154.608
C09708=1069.229,45.477,-67.369,172.758,25.422,154.607
C09709=1069.224,45.228,-67.353,172.756,25.419,154.607
C09710=1069.218,44.979,-67.337,172.755,25.416,154.607
C09711=1069.212,44.729,-67.321,172.754,25.413,154.606
C09712=1069.206,44.480,-67.304,172.752,25.411,154.606
C09713=1069.201,44.230,-67.288,172.751,25.408,154.606
C09714=1069.195,43.980,-67.272,172.750,25.405,154.605
C09715=1069.189,43.731,-67.256,172.748,25.403,154.605
C09716=1069.183,43.482,-67.239,172.747,25.400,154.605
C09717=1069.177,43.232,-67.223,172.746,25.397,154.604
C09718=1069.171,42.983,-67.207,172.744,25.395,154.604
C09719=1069.165,42.734,-67.191,172.743,25.392,154.603
C09720=1069.160,42.485,-67.175,172.741,25.390,154.603
C09721=1069.154,42.235,-67.159,172.740,25.387,154.603
C09722=1069.148,41.986,-67.143,172.738,25.384,154.602
C09723=1069.142,41.736,-67.127,172.736,25.381,154.602
C09724=1069.135,41.487,-67.111,172.735,25.378,154.602
C09725=1069.130,41.238,-67.095,172.734,25.376,154.601
C09726=1069.124,40.988,-67.079,172.732,25.373,154.601
C09727=1069.118,40.739,-67.063,172.731,25.370,154.601
C09728=1069.112,40.489,-67.047,172.730,25.368,154.600
C09729=1069.106,40.240,-67.031,172.728,25.365,154.600
C09730=1069.100,39.991,-67.014,172.727,25.363,154.600
C09731=1069.094,39.741,-66.999,172.725,25.360,154.599
C09732=1069.088,39.491,-66.983,172.724,25.357,154.599
C09733=1069.083,39.242,-66.966,172.723,25.355,154.599
C09734=1069.077,38.993,-66.950,172.721,25.352,154.598
C09735=1069.072,38.743,-66.935,172.720,25.349,154.598
C09736=1069.066,38.494,-66.919,172.719,25.346,154.598
C09737=1069.060,38.245,-66.902,172.717,25.344,154.597
C09738=1069.053,37.995,-66.887,172.716,25.341,154.597
C09739=1069.047,37.746,-66.871,172.715,25.338,154.596
C09740=1069.041,37.496,-66.855,172.713,25.336,154.596
C09741=1069.035,37.247,-66.839,172.712,25.333,154.596
C09742=1069.030,36.997,-66.823,172.710,25.331,154.596
C09743=1069.023,36.748,-66.807,172.709,25.328,154.595
C09744=1069.017,36.498,-66.792,172.708,25.326,154.595
C09745=1069.011,36.249,-66.776,172.706,25.323,154.594
C09746=1069.006,36.000,-66.760,172.705,25.320,154.594
C09747=1069.000,35.750,-66.745,172.704,25.317,154.594
C09748=1068.994,35.501,-66.728,172.702,25.315,154.594
C09749=1068.988,35.252,-66.712,172.701,25.312,154.593
C09750=1068.982,35.002,-66.697,172.699,25.310,154.593
C09751=1068.976,34.753,-66.681,172.698,25.307,154.592
C09752=1068.970,34.503,-66.665,172.697,25.304,154.592
C09753=1068.964,34.253,-66.649,172.695,25.302,154.592
C09754=1068.957,34.004,-66.634,172.694,25.299,154.591
C09755=1068.952,33.755,-66.618,172.693,25.296,154.591
C09756=1068.946,33.506,-66.602,172.691,25.294,154.591
C09757=1068.941,33.256,-66.587,172.690,25.291,154.590
C09758=1068.934,33.007,-66.571,172.689,25.288,154.590
C09759=1068.928,32.757,-66.555,172.687,25.286,154.590
C09760=1068.922,32.507,-66.539,172.686,25.283,154.589
C09761=1068.917,32.258,-66.525,172.683,25.280,154.589
C09762=1068.911,32.009,-66.508,172.682,25.277,154.589
C09763=1068.905,31.759,-66.493,172.681,25.275,154.588
C09764=1068.898,31.510,-66.477,172.679,25.272,154.588
C09765=1068.893,31.260,-66.462,172.678,25.270,154.588
C09766=1068.887,31.011,-66.445,172.677,25.267,154.587
C09767=1068.880,30.728,-66.428,172.675,25.264,154.587
C09768=1068.874,30.445,-66.410,172.674,25.261,154.587
C09769=1068.867,30.162,-66.393,172.673,25.258,154.586
C09770=1068.860,29.879,-66.374,172.671,25.255,154.586
C09771=1068.854,29.630,-66.359,172.669,25.252,154.585
C09772=1068.848,29.380,-66.344,172.668,25.250,154.585
C09773=1068.842,29.130,-66.328,172.666,25.247,154.585
C09774=1068.837,28.881,-66.313,172.665,25.245,154.584
C09775=1068.831,28.632,-66.297,172.664,25.242,154.584
C09776=1068.824,28.382,-66.282,172.662,25.239,154.584
C09777=1068.818,28.133,-66.266,172.661,25.236,154.583
C09778=1068.812,27.883,-66.251,172.660,25.234,154.583
C09779=1068.807,27.634,-66.235,172.658,25.231,154.583
C09780=1068.801,27.385,-66.219,172.657,25.229,154.582
C09781=1068.795,27.135,-66.204,172.656,25.226,154.582
C09782=1068.789,26.885,-66.189,172.654,25.224,154.582
C09783=1068.783,26.637,-66.173,172.653,25.221,154.581
C09784=1068.777,26.387,-66.158,172.651,25.218,154.581
C09785=1068.771,26.137,-66.143,172.650,25.215,154.581
C09786=1068.765,25.888,-66.127,172.649,25.213,154.580
C09787=1068.758,25.638,-66.112,172.647,25.210,154.580
C09788=1068.753,25.389,-66.097,172.646,25.208,154.580
C09789=1068.747,25.140,-66.081,172.644,25.206,154.579
C09790=1068.741,24.890,-66.065,172.643,25.203,154.579
C09791=1068.735,24.640,-66.050,172.642,25.200,154.579
C09792=1068.729,24.391,-66.036,172.640,25.197,154.578
C09793=1068.723,24.142,-66.020,172.639,25.195,154.578
C09794=1068.717,23.892,-66.005,172.638,25.192,154.578
C09795=1068.711,23.642,-65.989,172.636,25.190,154.577
C09796=1068.705,23.393,-65.974,172.635,25.187,154.577
C09797=1068.699,23.144,-65.958,172.634,25.185,154.577
C09798=1068.693,22.894,-65.943,172.632,25.182,154.576
C09799=1068.688,22.645,-65.928,172.631,25.179,154.576
C09800=1068.681,22.395,-65.913,172.630,25.176,154.576
C09801=1068.676,22.146,-65.898,172.628,25.174,154.575
C09802=1068.669,21.896,-65.882,172.627,25.172,154.575
C09803=1068.663,21.648,-65.867,172.625,25.169,154.575
C09804=1068.658,21.398,-65.852,172.624,25.166,154.574
C09805=1068.651,21.148,-65.837,172.623,25.163,154.574
C09806=1068.646,20.899,-65.822,172.621,25.161,154.574
C09807=1068.640,20.650,-65.806,172.619,25.158,154.573
C09808=1068.634,20.400,-65.790,172.618,25.156,154.573
C09809=1068.628,20.151,-65.776,172.616,25.153,154.573
C09810=1068.622,19.901,-65.761,172.615,25.150,154.572
C09811=1068.616,19.651,-65.745,172.614,25.147,154.572
C09812=1068.610,19.402,-65.731,172.612,25.145,154.572
C09813=1068.604,19.152,-65.716,172.611,25.143,154.571
C09814=1068.598,18.902,-65.700,172.609,25.140,154.571
C09815=1068.592,18.653,-65.685,172.608,25.137,154.571
C09816=1068.586,18.404,-65.670,172.607,25.135,154.570
C09817=1068.580,18.155,-65.655,172.605,25.132,154.570
C09818=1068.574,17.905,-65.640,172.604,25.130,154.570
C09819=1068.568,17.656,-65.625,172.603,25.127,154.569
C09820=1068.562,17.406,-65.610,172.601,25.125,154.569
C09821=1068.556,17.156,-65.595,172.600,25.122,154.569
C09822=1068.550,16.907,-65.580,172.598,25.119,154.569
C09823=1068.544,16.658,-65.565,172.597,25.116,154.568
C09824=1068.539,16.408,-65.550,172.596,25.114,154.568
C09825=1068.532,16.159,-65.535,172.594,25.112,154.568
C09826=1068.526,15.909,-65.520,172.593,25.109,154.567
C09827=1068.521,15.660,-65.505,172.592,25.106,154.567
C09828=1068.515,15.410,-65.490,172.590,25.104,154.566
C09829=1068.508,15.160,-65.475,172.589,25.101,154.566
C09830=1068.502,14.912,-65.460,172.587,25.099,154.566
C09831=1068.496,14.629,-65.444,172.586,25.096,154.566
C09832=1068.489,14.349,-65.427,172.584,25.093,154.565
C09833=1068.482,14.066,-65.410,172.583,25.090,154.565
C09834=1068.475,13.785,-65.392,172.581,25.087,154.564
C09835=1068.470,13.535,-65.379,172.580,25.084,154.564
C09836=1068.463,13.286,-65.364,172.579,25.082,154.564
C09837=1068.457,13.036,-65.349,172.577,25.080,154.564
C09838=1068.451,12.787,-65.334,172.576,25.077,154.563
C09839=1068.445,12.537,-65.319,172.574,25.074,154.563
C09840=1068.438,12.288,-65.304,172.573,25.072,154.563
C09841=1068.433,12.039,-65.289,172.572,25.069,154.562
C09842=1068.427,11.789,-65.274,172.570,25.067,154.562
C09843=1068.421,11.540,-65.260,172.569,25.065,154.562
C09844=1068.415,11.290,-65.245,172.568,25.062,154.561
C09845=1068.409,11.040,-65.230,172.566,25.059,154.561
C09846=1068.403,10.791,-65.216,172.565,25.057,154.561
C09847=1068.397,10.541,-65.201,172.563,25.055,154.560
C09848=1068.391,10.292,-65.186,172.562,25.052,154.560
C09849=1068.384,10.043,-65.171,172.561,25.049,154.560
C09850=1068.378,9.792,-65.157,172.559,25.047,154.559
C09851=1068.373,9.544,-65.142,172.558,25.044,154.559
C09852=1068.366,9.294,-65.128,172.556,25.042,154.559
C09853=1068.360,9.045,-65.113,172.555,25.039,154.559
C09854=1068.354,8.795,-65.098,172.553,25.036,154.558
C09855=1068.348,8.545,-65.084,172.551,25.034,154.558
C09856=1068.342,8.296,-65.069,172.550,25.031,154.558
C09857=1068.336,8.046,-65.054,172.549,25.029,154.557
C09858=1068.330,7.797,-65.040,172.547,25.026,154.557
C09859=1068.324,7.547,-65.025,172.546,25.024,154.557
C09860=1068.318,7.298,-65.011,172.544,25.021,154.556
C09861=1068.312,7.049,-64.996,172.543,25.018,154.556
C09862=1068.306,6.799,-64.982,172.542,25.016,154.556
C09863=1068.300,6.549,-64.967,172.540,25.014,154.555
C09864=1068.294,6.300,-64.953,172.539,25.011,154.555
C09865=1068.288,6.051,-64.938,172.538,25.008,154.555
C09866=1068.282,5.801,-64.924,172.536,25.006,154.555
C09867=1068.276,5.551,-64.909,172.535,25.004,154.554
C09868=1068.270,5.303,-64.894,172.534,25.001,154.554
C09869=1068.264,5.052,-64.880,172.532,24.998,154.554
C09870=1068.258,4.803,-64.865,172.531,24.996,154.553
C09871=1068.252,4.554,-64.850,172.529,24.993,154.553
C09872=1068.246,4.304,-64.837,172.528,24.991,154.553
C09873=1068.240,4.054,-64.822,172.527,24.988,154.552
C09874=1068.234,3.805,-64.808,172.525,24.986,154.552
C09875=1068.228,3.555,-64.793,172.524,24.983,154.552
C09876=1068.222,3.306,-64.778,172.522,24.981,154.551
C09877=1068.216,3.056,-64.764,172.521,24.978,154.551
C09878=1068.210,2.807,-64.749,172.520,24.976,154.551
C09879=1068.204,2.557,-64.734,172.518,24.973,154.550
C09880=1068.199,2.308,-64.721,172.517,24.971,154.550
C09881=1068.193,2.059,-64.706,172.516,24.968,154.550
C09882=1068.187,1.808,-64.692,172.514,24.966,154.550
C09883=1068.181,1.560,-64.677,172.513,24.963,154.549
C09884=1068.175,1.309,-64.663,172.511,24.961,154.549
C09885=1068.169,1.060,-64.648,172.510,24.958,154.549
C09886=1068.163,0.810,-64.634,172.509,24.956,154.548
C09887=1068.157,0.561,-64.620,172.507,24.953,154.548
C09888=1068.152,0.312,-64.606,172.506,24.951,154.548
C09889=1068.145,0.062,-64.591,172.505,24.948,154.547
C09890=1068.140,-0.188,-64.577,172.503,24.945,154.547
C09891=1068.134,-0.437,-64.562,172.502,24.943,154.547
C09892=1068.128,-0.687,-64.548,172.501,24.940,154.546
C09893=1068.122,-0.936,-64.534,172.499,24.938,154.546
C09894=1068.116,-1.186,-64.519,172.498,24.935,154.546
C09895=1068.109,-1.466,-64.504,172.495,24.932,154.546
C09896=1068.103,-1.745,-64.488,172.494,24.930,154.545
C09897=1068.096,-2.024,-64.472,172.493,24.927,154.545
C09898=1068.090,-2.304,-64.456,172.491,24.924,154.544
C09899=1068.084,-2.553,-64.441,172.489,24.921,154.544
C09900=1068.078,-2.803,-64.427,172.488,24.919,154.544
C09901=1068.072,-3.052,-64.413,172.487,24.916,154.544
C09902=1068.066,-3.302,-64.399,172.485,24.914,154.543
C09903=1068.060,-3.552,-64.384,172.484,24.911,154.543
C09904=1068.054,-3.801,-64.370,172.482,24.909,154.543
C09905=1068.048,-4.051,-64.356,172.481,24.907,154.542
C09906=1068.042,-4.300,-64.342,172.479,24.904,154.542
C09907=1068.035,-4.550,-64.328,172.478,24.902,154.542
C09908=1068.030,-4.800,-64.314,172.477,24.899,154.542
C09909=1068.024,-5.049,-64.300,172.475,24.897,154.541
C09910=1068.017,-5.299,-64.286,172.474,24.894,154.541
C09911=1068.012,-5.548,-64.272,172.473,24.892,154.541
C09912=1068.006,-5.797,-64.257,172.471,24.889,154.540
C09913=1067.999,-6.047,-64.244,172.470,24.887,154.540
C09914=1067.994,-6.297,-64.230,172.468,24.885,154.540
C09915=1067.987,-6.546,-64.215,172.467,24.882,154.540
C09916=1067.981,-6.796,-64.202,172.465,24.880,154.539
C09917=1067.975,-7.045,-64.188,172.464,24.877,154.539
C09918=1067.969,-7.295,-64.174,172.463,24.875,154.539
C09919=1067.963,-7.544,-64.160,172.461,24.872,154.538
C09920=1067.957,-7.794,-64.146,172.460,24.870,154.538
C09921=1067.951,-8.044,-64.132,172.459,24.868,154.538
C09922=1067.945,-8.293,-64.118,172.457,24.865,154.538
C09923=1067.939,-8.542,-64.104,172.456,24.863,154.537
C09924=1067.932,-8.792,-64.090,172.454,24.860,154.537
C09925=1067.927,-9.042,-64.076,172.453,24.858,154.537
C09926=1067.921,-9.291,-64.063,172.452,24.856,154.536
C09927=1067.914,-9.541,-64.048,172.450,24.853,154.536
C09928=1067.909,-9.790,-64.034,172.449,24.850,154.536
C09929=1067.903,-10.039,-64.021,172.447,24.848,154.536
C09930=1067.897,-10.290,-64.007,172.446,24.846,154.535
C09931=1067.891,-10.539,-63.993,172.444,24.843,154.535
C09932=1067.885,-10.788,-63.979,172.442,24.841,154.535
C09933=1067.879,-11.038,-63.965,172.441,24.838,154.534
C09934=1067.872,-11.288,-63.951,172.439,24.836,154.534
C09935=1067.867,-11.537,-63.937,172.438,24.834,154.534
C09936=1067.861,-11.787,-63.924,172.437,24.831,154.534
C09937=1067.855,-12.036,-63.910,172.435,24.829,154.533
C09938=1067.849,-12.286,-63.896,172.434,24.826,154.533
C09939=1067.843,-12.535,-63.882,172.433,24.824,154.533
C09940=1067.837,-12.784,-63.868,172.431,24.821,154.532
C09941=1067.831,-13.034,-63.855,172.430,24.819,154.532
C09942=1067.825,-13.284,-63.841,172.428,24.816,154.532
C09943=1067.819,-13.534,-63.827,172.427,24.814,154.532
C09944=1067.813,-13.783,-63.814,172.426,24.812,154.531
C09945=1067.808,-14.032,-63.800,172.424,24.809,154.531
C09946=1067.801,-14.282,-63.786,172.423,24.807,154.531
C09947=1067.795,-14.532,-63.772,172.421,24.805,154.531
C09948=1067.789,-14.781,-63.759,172.420,24.802,154.530
C09949=1067.784,-15.031,-63.745,172.419,24.800,154.530
C09950=1067.777,-15.281,-63.731,172.417,24.797,154.530
C09951=1067.771,-15.530,-63.718,172.416,24.795,154.529
C09952=1067.765,-15.780,-63.704,172.414,24.793,154.529
C09953=1067.760,-16.029,-63.690,172.413,24.790,154.529
C09954=1067.753,-16.279,-63.677,172.412,24.788,154.529
C09955=1067.747,-16.528,-63.664,172.410,24.786,154.528
C09956=1067.741,-16.778,-63.650,172.409,24.783,154.528
C09957=1067.735,-17.027,-63.636,172.407,24.781,154.528
C09958=1067.728,-17.277,-63.623,172.406,24.778,154.528
C09959=1067.722,-17.555,-63.607,172.404,24.776,154.527
C09960=1067.715,-17.833,-63.592,172.402,24.773,154.527
C09961=1067.709,-18.111,-63.577,172.401,24.771,154.527
C09962=1067.701,-18.388,-63.563,172.399,24.768,154.526
C09963=1067.695,-18.639,-63.548,172.397,24.765,154.526
C09964=1067.689,-18.888,-63.535,172.396,24.763,154.526
C09965=1067.683,-19.137,-63.522,172.394,24.761,154.526
C09966=1067.678,-19.387,-63.508,172.393,24.759,154.525
C09967=1067.672,-19.637,-63.495,172.391,24.756,154.525
C09968=1067.665,-19.887,-63.482,172.390,24.754,154.525
C09969=1067.659,-20.136,-63.468,172.389,24.752,154.525
C09970=1067.653,-20.386,-63.455,172.387,24.749,154.524
C09971=1067.647,-20.635,-63.441,172.386,24.747,154.524
C09972=1067.641,-20.884,-63.427,172.384,24.745,154.524
C09973=1067.635,-21.134,-63.414,172.383,24.742,154.524
C09974=1067.629,-21.384,-63.401,172.382,24.740,154.523
C09975=1067.623,-21.634,-63.387,172.380,24.737,154.523
C09976=1067.617,-21.883,-63.374,172.379,24.735,154.523
C09977=1067.611,-22.132,-63.361,172.377,24.733,154.523
C09978=1067.605,-22.382,-63.347,172.376,24.731,154.522
C09979=1067.599,-22.631,-63.334,172.375,24.728,154.522
C09980=1067.593,-22.881,-63.321,172.373,24.726,154.522
C09981=1067.587,-23.131,-63.307,172.372,24.724,154.522
C09982=1067.581,-23.381,-63.294,172.370,24.721,154.521
C09983=1067.575,-23.630,-63.280,172.369,24.719,154.521
C09984=1067.569,-23.880,-63.268,172.368,24.717,154.521
C09985=1067.563,-24.129,-63.254,172.366,24.714,154.520
C09986=1067.557,-24.379,-63.241,172.365,24.712,154.520
C09987=1067.551,-24.628,-63.227,172.363,24.710,154.520
C09988=1067.546,-24.878,-63.214,172.361,24.707,154.520
C09989=1067.539,-25.127,-63.201,172.359,24.705,154.520
C09990=1067.533,-25.377,-63.188,172.358,24.703,154.519
C09991=1067.526,-25.627,-63.174,172.357,24.700,154.519
C09992=1067.521,-25.877,-63.161,172.355,24.698,154.519
C09993=1067.515,-26.126,-63.148,172.354,24.695,154.518
C09994=1067.509,-26.375,-63.134,172.352,24.694,154.518
C09995=1067.503,-26.625,-63.122,172.351,24.691,154.518
C09996=1067.497,-26.875,-63.108,172.350,24.689,154.518
//INST
///DATE 2021/06/17 10:55
///ATTR SC,RW,RJ
////FRAME ROBOT
///GROUP1 RB1
NOP
MOVL C00000 V=800.0 PL=0
MOVL C00001 V=800.0 PL=0
MOVL C00002 V=800.0 PL=0
MOVL C00003 V=800.0 PL=0
MOVL C00004 V=800.0 PL=0
MOVL C00005 V=800.0 PL=0
MOVL C00006 V=800.0 PL=0
MOVL C00007 V=800.0 PL=0
MOVL C00008 V=800.0 PL=0
MOVL C00009 V=800.0 PL=0
MOVL C00010 V=800.0 PL=0
MOVL C00011 V=800.0 PL=0
MOVL C00012 V=800.0 PL=0
MOVL C00013 V=800.0 PL=0
MOVL C00014 V=800.0 PL=0
MOVL C00015 V=800.0 PL=0
MOVL C00016 V=800.0 PL=0
MOVL C00017 V=800.0 PL=0
MOVL C00018 V=800.0 PL=0
MOVL C00019 V=800.0 PL=0
MOVL C00020 V=800.0 PL=0
MOVL C00021 V=800.0 PL=0
MOVL C00022 V=800.0 PL=0
MOVL C00023 V=800.0 PL=0
MOVL C00024 V=800.0 PL=0
MOVL C00025 V=800.0 PL=0
MOVL C00026 V=800.0 PL=0
MOVL C00027 V=800.0 PL=0
MOVL C00028 V=800.0 PL=0
MOVL C00029 V=800.0 PL=0
MOVL C00030 V=800.0 PL=0
MOVL C00031 V=800.0 PL=0
MOVL C00032 V=800.0 PL=0
MOVL C00033 V=800.0 PL=0
MOVL C00034 V=800.0 PL=0
MOVL C00035 V=800.0 PL=0
MOVL C00036 V=800.0 PL=0
MOVL C00037 V=800.0 PL=0
MOVL C00038 V=800.0 PL=0
MOVL C00039 V=800.0 PL=0
MOVL C00040 V=800.0 PL=0
MOVL C00041 V=800.0 PL=0
MOVL C00042 V=800.0 PL=0
MOVL C00043 V=800.0 PL=0
MOVL C00044 V=800.0 PL=0
MOVL C00045 V=800.0 PL=0
MOVL C00046 V=800.0 PL=0
MOVL C00047 V=800.0 PL=0
MOVL C00048 V=800.0 PL=0
MOVL C00049 V=800.0 PL=0
MOVL C00050 V=800.0 PL=0
MOVL C00051 V=800.0 PL=0
MOVL C00052 V=800.0 PL=0
MOVL C00053 V=800.0 PL=0
MOVL C00054 V=800.0 PL=0
MOVL C00055 V=800.0 PL=0
MOVL C00056 V=800.0 PL=0
MOVL C00057 V=800.0 PL=0
MOVL C00058 V=800.0 PL=0
MOVL C00059 V=800.0 PL=0
MOVL C00060 V=800.0 PL=0
MOVL C00061 V=800.0 PL=0
MOVL C00062 V=800.0 PL=0
MOVL C00063 V=800.0 PL=0
MOVL C00064 V=800.0 PL=0
MOVL C00065 V=800.0 PL=0
MOVL C00066 V=800.0 PL=0
MOVL C00067 V=800.0 PL=0
MOVL C00068 V=800.0 PL=0
MOVL C00069 V=800.0 PL=0
MOVL C00070 V=800.0 PL=0
MOVL C00071 V=800.0 PL=0
MOVL C00072 V=800.0 PL=0
MOVL C00073 V=800.0 PL=0
MOVL C00074 V=800.0 PL=0
MOVL C00075 V=800.0 PL=0
MOVL C00076 V=800.0 PL=0
MOVL C00077 V=800.0 PL=0
MOVL C00078 V=800.0 PL=0
MOVL C00079 V=800.0 PL=0
MOVL C00080 V=800.0 PL=0
MOVL C00081 V=800.0 PL=0
MOVL C00082 V=800.0 PL=0
MOVL C00083 V=800.0 PL=0
MOVL C00084 V=800.0 PL=0
MOVL C00085 V=800.0 PL=0
MOVL C00086 V=800.0 PL=0
MOVL C00087 V=800.0 PL=0
MOVL C00088 V=800.0 PL=0
MOVL C00089 V=800.0 PL=0
MOVL C00090 V=800.0 PL=0
MOVL C00091 V=800.0 PL=0
MOVL C00092 V=800.0 PL=0
MOVL C00093 V=800.0 PL=0
MOVL C00094 V=800.0 PL=0
MOVL C00095 V=800.0 PL=0
MOVL C00096 V=800.0 PL=0
MOVL C00097 V=800.0 PL=0
MOVL C00098 V=800.0 PL=0
MOVL C00099 V=800.0 PL=0
MOVL C00100 V=800.0 PL=0
MOVL C00101 V=800.0 PL=0
MOVL C00102 V=800.0 PL=0
MOVL C00103 V=800.0 PL=0
MOVL C00104 V=800.0 PL=0
MOVL C00105 V=800.0 PL=0
MOVL C00106 V=800.0 PL=0
MOVL C00107 V=800.0 PL=0
MOVL C00108 V=800.0 PL=0
MOVL C00109 V=800.0 PL=0
MOVL C00110 V=800.0 PL=0
MOVL C00111 V=800.0 PL=0
MOVL C00112 V=800.0 PL=0
MOVL C00113 V=800.0 PL=0
MOVL C00114 V=800.0 PL=0
MOVL C00115 V=800.0 PL=0
MOVL C00116 V=800.0 PL=0
MOVL C00117 V=800.0 PL=0
MOVL C00118 V=800.0 PL=0
MOVL C00119 V=800.0 PL=0
MOVL C00120 V=800.0 PL=0
MOVL C00121 V=800.0 PL=0
MOVL C00122 V=800.0 PL=0
MOVL C00123 V=800.0 PL=0
MOVL C00124 V=800.0 PL=0
MOVL C00125 V=800.0 PL=0
MOVL C00126 V=800.0 PL=0
MOVL C00127 V=800.0 PL=0
MOVL C00128 V=800.0 PL=0
MOVL C00129 V=800.0 PL=0
MOVL C00130 V=800.0 PL=0
MOVL C00131 V=800.0 PL=0
MOVL C00132 V=800.0 PL=0
MOVL C00133 V=800.0 PL=0
MOVL C00134 V=800.0 PL=0
MOVL C00135 V=800.0 PL=0
MOVL C00136 V=800.0 PL=0
MOVL C00137 V=800.0 PL=0
MOVL C00138 V=800.0 PL=0
MOVL C00139 V=800.0 PL=0
MOVL C00140 V=800.0 PL=0
MOVL C00141 V=800.0 PL=0
MOVL C00142 V=800.0 PL=0
MOVL C00143 V=800.0 PL=0
MOVL C00144 V=800.0 PL=0
MOVL C00145 V=800.0 PL=0
MOVL C00146 V=800.0 PL=0
MOVL C00147 V=800.0 PL=0
MOVL C00148 V=800.0 PL=0
MOVL C00149 V=800.0 PL=0
MOVL C00150 V=800.0 PL=0
MOVL C00151 V=800.0 PL=0
MOVL C00152 V=800.0 PL=0
MOVL C00153 V=800.0 PL=0
MOVL C00154 V=800.0 PL=0
MOVL C00155 V=800.0 PL=0
MOVL C00156 V=800.0 PL=0
MOVL C00157 V=800.0 PL=0
MOVL C00158 V=800.0 PL=0
MOVL C00159 V=800.0 PL=0
MOVL C00160 V=800.0 PL=0
MOVL C00161 V=800.0 PL=0
MOVL C00162 V=800.0 PL=0
MOVL C00163 V=800.0 PL=0
MOVL C00164 V=800.0 PL=0
MOVL C00165 V=800.0 PL=0
MOVL C00166 V=800.0 PL=0
MOVL C00167 V=800.0 PL=0
MOVL C00168 V=800.0 PL=0
MOVL C00169 V=800.0 PL=0
MOVL C00170 V=800.0 PL=0
MOVL C00171 V=800.0 PL=0
MOVL C00172 V=800.0 PL=0
MOVL C00173 V=800.0 PL=0
MOVL C00174 V=800.0 PL=0
MOVL C00175 V=800.0 PL=0
MOVL C00176 V=800.0 PL=0
MOVL C00177 V=800.0 PL=0
MOVL C00178 V=800.0 PL=0
MOVL C00179 V=800.0 PL=0
MOVL C00180 V=800.0 PL=0
MOVL C00181 V=800.0 PL=0
MOVL C00182 V=800.0 PL=0
MOVL C00183 V=800.0 PL=0
MOVL C00184 V=800.0 PL=0
MOVL C00185 V=800.0 PL=0
MOVL C00186 V=800.0 PL=0
MOVL C00187 V=800.0 PL=0
MOVL C00188 V=800.0 PL=0
MOVL C00189 V=800.0 PL=0
MOVL C00190 V=800.0 PL=0
MOVL C00191 V=800.0 PL=0
MOVL C00192 V=800.0 PL=0
MOVL C00193 V=800.0 PL=0
MOVL C00194 V=800.0 PL=0
MOVL C00195 V=800.0 PL=0
MOVL C00196 V=800.0 PL=0
MOVL C00197 V=800.0 PL=0
MOVL C00198 V=800.0 PL=0
MOVL C00199 V=800.0 PL=0
MOVL C00200 V=800.0 PL=0
MOVL C00201 V=800.0 PL=0
MOVL C00202 V=800.0 PL=0
MOVL C00203 V=800.0 PL=0
MOVL C00204 V=800.0 PL=0
MOVL C00205 V=800.0 PL=0
MOVL C00206 V=800.0 PL=0
MOVL C00207 V=800.0 PL=0
MOVL C00208 V=800.0 PL=0
MOVL C00209 V=800.0 PL=0
MOVL C00210 V=800.0 PL=0
MOVL C00211 V=800.0 PL=0
MOVL C00212 V=800.0 PL=0
MOVL C00213 V=800.0 PL=0
MOVL C00214 V=800.0 PL=0
MOVL C00215 V=800.0 PL=0
MOVL C00216 V=800.0 PL=0
MOVL C00217 V=800.0 PL=0
MOVL C00218 V=800.0 PL=0
MOVL C00219 V=800.0 PL=0
MOVL C00220 V=800.0 PL=0
MOVL C00221 V=800.0 PL=0
MOVL C00222 V=800.0 PL=0
MOVL C00223 V=800.0 PL=0
MOVL C00224 V=800.0 PL=0
MOVL C00225 V=800.0 PL=0
MOVL C00226 V=800.0 PL=0
MOVL C00227 V=800.0 PL=0
MOVL C00228 V=800.0 PL=0
MOVL C00229 V=800.0 PL=0
MOVL C00230 V=800.0 PL=0
MOVL C00231 V=800.0 PL=0
MOVL C00232 V=800.0 PL=0
MOVL C00233 V=800.0 PL=0
MOVL C00234 V=800.0 PL=0
MOVL C00235 V=800.0 PL=0
MOVL C00236 V=800.0 PL=0
MOVL C00237 V=800.0 PL=0
MOVL C00238 V=800.0 PL=0
MOVL C00239 V=800.0 PL=0
MOVL C00240 V=800.0 PL=0
MOVL C00241 V=800.0 PL=0
MOVL C00242 V=800.0 PL=0
MOVL C00243 V=800.0 PL=0
MOVL C00244 V=800.0 PL=0
MOVL C00245 V=800.0 PL=0
MOVL C00246 V=800.0 PL=0
MOVL C00247 V=800.0 PL=0
MOVL C00248 V=800.0 PL=0
MOVL C00249 V=800.0 PL=0
MOVL C00250 V=800.0 PL=0
MOVL C00251 V=800.0 PL=0
MOVL C00252 V=800.0 PL=0
MOVL C00253 V=800.0 PL=0
MOVL C00254 V=800.0 PL=0
MOVL C00255 V=800.0 PL=0
MOVL C00256 V=800.0 PL=0
MOVL C00257 V=800.0 PL=0
MOVL C00258 V=800.0 PL=0
MOVL C00259 V=800.0 PL=0
MOVL C00260 V=800.0 PL=0
MOVL C00261 V=800.0 PL=0
MOVL C00262 V=800.0 PL=0
MOVL C00263 V=800.0 PL=0
MOVL C00264 V=800.0 PL=0
MOVL C00265 V=800.0 PL=0
MOVL C00266 V=800.0 PL=0
MOVL C00267 V=800.0 PL=0
MOVL C00268 V=800.0 PL=0
MOVL C00269 V=800.0 PL=0
MOVL C00270 V=800.0 PL=0
MOVL C00271 V=800.0 PL=0
MOVL C00272 V=800.0 PL=0
MOVL C00273 V=800.0 PL=0
MOVL C00274 V=800.0 PL=0
MOVL C00275 V=800.0 PL=0
MOVL C00276 V=800.0 PL=0
MOVL C00277 V=800.0 PL=0
MOVL C00278 V=800.0 PL=0
MOVL C00279 V=800.0 PL=0
MOVL C00280 V=800.0 PL=0
MOVL C00281 V=800.0 PL=0
MOVL C00282 V=800.0 PL=0
MOVL C00283 V=800.0 PL=0
MOVL C00284 V=800.0 PL=0
MOVL C00285 V=800.0 PL=0
MOVL C00286 V=800.0 PL=0
MOVL C00287 V=800.0 PL=0
MOVL C00288 V=800.0 PL=0
MOVL C00289 V=800.0 PL=0
MOVL C00290 V=800.0 PL=0
MOVL C00291 V=800.0 PL=0
MOVL C00292 V=800.0 PL=0
MOVL C00293 V=800.0 PL=0
MOVL C00294 V=800.0 PL=0
MOVL C00295 V=800.0 PL=0
MOVL C00296 V=800.0 PL=0
MOVL C00297 V=800.0 PL=0
MOVL C00298 V=800.0 PL=0
MOVL C00299 V=800.0 PL=0
MOVL C00300 V=800.0 PL=0
MOVL C00301 V=800.0 PL=0
MOVL C00302 V=800.0 PL=0
MOVL C00303 V=800.0 PL=0
MOVL C00304 V=800.0 PL=0
MOVL C00305 V=800.0 PL=0
MOVL C00306 V=800.0 PL=0
MOVL C00307 V=800.0 PL=0
MOVL C00308 V=800.0 PL=0
MOVL C00309 V=800.0 PL=0
MOVL C00310 V=800.0 PL=0
MOVL C00311 V=800.0 PL=0
MOVL C00312 V=800.0 PL=0
MOVL C00313 V=800.0 PL=0
MOVL C00314 V=800.0 PL=0
MOVL C00315 V=800.0 PL=0
MOVL C00316 V=800.0 PL=0
MOVL C00317 V=800.0 PL=0
MOVL C00318 V=800.0 PL=0
MOVL C00319 V=800.0 PL=0
MOVL C00320 V=800.0 PL=0
MOVL C00321 V=800.0 PL=0
MOVL C00322 V=800.0 PL=0
MOVL C00323 V=800.0 PL=0
MOVL C00324 V=800.0 PL=0
MOVL C00325 V=800.0 PL=0
MOVL C00326 V=800.0 PL=0
MOVL C00327 V=800.0 PL=0
MOVL C00328 V=800.0 PL=0
MOVL C00329 V=800.0 PL=0
MOVL C00330 V=800.0 PL=0
MOVL C00331 V=800.0 PL=0
MOVL C00332 V=800.0 PL=0
MOVL C00333 V=800.0 PL=0
MOVL C00334 V=800.0 PL=0
MOVL C00335 V=800.0 PL=0
MOVL C00336 V=800.0 PL=0
MOVL C00337 V=800.0 PL=0
MOVL C00338 V=800.0 PL=0
MOVL C00339 V=800.0 PL=0
MOVL C00340 V=800.0 PL=0
MOVL C00341 V=800.0 PL=0
MOVL C00342 V=800.0 PL=0
MOVL C00343 V=800.0 PL=0
MOVL C00344 V=800.0 PL=0
MOVL C00345 V=800.0 PL=0
MOVL C00346 V=800.0 PL=0
MOVL C00347 V=800.0 PL=0
MOVL C00348 V=800.0 PL=0
MOVL C00349 V=800.0 PL=0
MOVL C00350 V=800.0 PL=0
MOVL C00351 V=800.0 PL=0
MOVL C00352 V=800.0 PL=0
MOVL C00353 V=800.0 PL=0
MOVL C00354 V=800.0 PL=0
MOVL C00355 V=800.0 PL=0
MOVL C00356 V=800.0 PL=0
MOVL C00357 V=800.0 PL=0
MOVL C00358 V=800.0 PL=0
MOVL C00359 V=800.0 PL=0
MOVL C00360 V=800.0 PL=0
MOVL C00361 V=800.0 PL=0
MOVL C00362 V=800.0 PL=0
MOVL C00363 V=800.0 PL=0
MOVL C00364 V=800.0 PL=0
MOVL C00365 V=800.0 PL=0
MOVL C00366 V=800.0 PL=0
MOVL C00367 V=800.0 PL=0
MOVL C00368 V=800.0 PL=0
MOVL C00369 V=800.0 PL=0
MOVL C00370 V=800.0 PL=0
MOVL C00371 V=800.0 PL=0
MOVL C00372 V=800.0 PL=0
MOVL C00373 V=800.0 PL=0
MOVL C00374 V=800.0 PL=0
MOVL C00375 V=800.0 PL=0
MOVL C00376 V=800.0 PL=0
MOVL C00377 V=800.0 PL=0
MOVL C00378 V=800.0 PL=0
MOVL C00379 V=800.0 PL=0
MOVL C00380 V=800.0 PL=0
MOVL C00381 V=800.0 PL=0
MOVL C00382 V=800.0 PL=0
MOVL C00383 V=800.0 PL=0
MOVL C00384 V=800.0 PL=0
MOVL C00385 V=800.0 PL=0
MOVL C00386 V=800.0 PL=0
MOVL C00387 V=800.0 PL=0
MOVL C00388 V=800.0 PL=0
MOVL C00389 V=800.0 PL=0
MOVL C00390 V=800.0 PL=0
MOVL C00391 V=800.0 PL=0
MOVL C00392 V=800.0 PL=0
MOVL C00393 V=800.0 PL=0
MOVL C00394 V=800.0 PL=0
MOVL C00395 V=800.0 PL=0
MOVL C00396 V=800.0 PL=0
MOVL C00397 V=800.0 PL=0
MOVL C00398 V=800.0 PL=0
MOVL C00399 V=800.0 PL=0
MOVL C00400 V=800.0 PL=0
MOVL C00401 V=800.0 PL=0
MOVL C00402 V=800.0 PL=0
MOVL C00403 V=800.0 PL=0
MOVL C00404 V=800.0 PL=0
MOVL C00405 V=800.0 PL=0
MOVL C00406 V=800.0 PL=0
MOVL C00407 V=800.0 PL=0
MOVL C00408 V=800.0 PL=0
MOVL C00409 V=800.0 PL=0
MOVL C00410 V=800.0 PL=0
MOVL C00411 V=800.0 PL=0
MOVL C00412 V=800.0 PL=0
MOVL C00413 V=800.0 PL=0
MOVL C00414 V=800.0 PL=0
MOVL C00415 V=800.0 PL=0
MOVL C00416 V=800.0 PL=0
MOVL C00417 V=800.0 PL=0
MOVL C00418 V=800.0 PL=0
MOVL C00419 V=800.0 PL=0
MOVL C00420 V=800.0 PL=0
MOVL C00421 V=800.0 PL=0
MOVL C00422 V=800.0 PL=0
MOVL C00423 V=800.0 PL=0
MOVL C00424 V=800.0 PL=0
MOVL C00425 V=800.0 PL=0
MOVL C00426 V=800.0 PL=0
MOVL C00427 V=800.0 PL=0
MOVL C00428 V=800.0 PL=0
MOVL C00429 V=800.0 PL=0
MOVL C00430 V=800.0 PL=0
MOVL C00431 V=800.0 PL=0
MOVL C00432 V=800.0 PL=0
MOVL C00433 V=800.0 PL=0
MOVL C00434 V=800.0 PL=0
MOVL C00435 V=800.0 PL=0
MOVL C00436 V=800.0 PL=0
MOVL C00437 V=800.0 PL=0
MOVL C00438 V=800.0 PL=0
MOVL C00439 V=800.0 PL=0
MOVL C00440 V=800.0 PL=0
MOVL C00441 V=800.0 PL=0
MOVL C00442 V=800.0 PL=0
MOVL C00443 V=800.0 PL=0
MOVL C00444 V=800.0 PL=0
MOVL C00445 V=800.0 PL=0
MOVL C00446 V=800.0 PL=0
MOVL C00447 V=800.0 PL=0
MOVL C00448 V=800.0 PL=0
MOVL C00449 V=800.0 PL=0
MOVL C00450 V=800.0 PL=0
MOVL C00451 V=800.0 PL=0
MOVL C00452 V=800.0 PL=0
MOVL C00453 V=800.0 PL=0
MOVL C00454 V=800.0 PL=0
MOVL C00455 V=800.0 PL=0
MOVL C00456 V=800.0 PL=0
MOVL C00457 V=800.0 PL=0
MOVL C00458 V=800.0 PL=0
MOVL C00459 V=800.0 PL=0
MOVL C00460 V=800.0 PL=0
MOVL C00461 V=800.0 PL=0
MOVL C00462 V=800.0 PL=0
MOVL C00463 V=800.0 PL=0
MOVL C00464 V=800.0 PL=0
MOVL C00465 V=800.0 PL=0
MOVL C00466 V=800.0 PL=0
MOVL C00467 V=800.0 PL=0
MOVL C00468 V=800.0 PL=0
MOVL C00469 V=800.0 PL=0
MOVL C00470 V=800.0 PL=0
MOVL C00471 V=800.0 PL=0
MOVL C00472 V=800.0 PL=0
MOVL C00473 V=800.0 PL=0
MOVL C00474 V=800.0 PL=0
MOVL C00475 V=800.0 PL=0
MOVL C00476 V=800.0 PL=0
MOVL C00477 V=800.0 PL=0
MOVL C00478 V=800.0 PL=0
MOVL C00479 V=800.0 PL=0
MOVL C00480 V=800.0 PL=0
MOVL C00481 V=800.0 PL=0
MOVL C00482 V=800.0 PL=0
MOVL C00483 V=800.0 PL=0
MOVL C00484 V=800.0 PL=0
MOVL C00485 V=800.0 PL=0
MOVL C00486 V=800.0 PL=0
MOVL C00487 V=800.0 PL=0
MOVL C00488 V=800.0 PL=0
MOVL C00489 V=800.0 PL=0
MOVL C00490 V=800.0 PL=0
MOVL C00491 V=800.0 PL=0
MOVL C00492 V=800.0 PL=0
MOVL C00493 V=800.0 PL=0
MOVL C00494 V=800.0 PL=0
MOVL C00495 V=800.0 PL=0
MOVL C00496 V=800.0 PL=0
MOVL C00497 V=800.0 PL=0
MOVL C00498 V=800.0 PL=0
MOVL C00499 V=800.0 PL=0
MOVL C00500 V=800.0 PL=0
MOVL C00501 V=800.0 PL=0
MOVL C00502 V=800.0 PL=0
MOVL C00503 V=800.0 PL=0
MOVL C00504 V=800.0 PL=0
MOVL C00505 V=800.0 PL=0
MOVL C00506 V=800.0 PL=0
MOVL C00507 V=800.0 PL=0
MOVL C00508 V=800.0 PL=0
MOVL C00509 V=800.0 PL=0
MOVL C00510 V=800.0 PL=0
MOVL C00511 V=800.0 PL=0
MOVL C00512 V=800.0 PL=0
MOVL C00513 V=800.0 PL=0
MOVL C00514 V=800.0 PL=0
MOVL C00515 V=800.0 PL=0
MOVL C00516 V=800.0 PL=0
MOVL C00517 V=800.0 PL=0
MOVL C00518 V=800.0 PL=0
MOVL C00519 V=800.0 PL=0
MOVL C00520 V=800.0 PL=0
MOVL C00521 V=800.0 PL=0
MOVL C00522 V=800.0 PL=0
MOVL C00523 V=800.0 PL=0
MOVL C00524 V=800.0 PL=0
MOVL C00525 V=800.0 PL=0
MOVL C00526 V=800.0 PL=0
MOVL C00527 V=800.0 PL=0
MOVL C00528 V=800.0 PL=0
MOVL C00529 V=800.0 PL=0
MOVL C00530 V=800.0 PL=0
MOVL C00531 V=800.0 PL=0
MOVL C00532 V=800.0 PL=0
MOVL C00533 V=800.0 PL=0
MOVL C00534 V=800.0 PL=0
MOVL C00535 V=800.0 PL=0
MOVL C00536 V=800.0 PL=0
MOVL C00537 V=800.0 PL=0
MOVL C00538 V=800.0 PL=0
MOVL C00539 V=800.0 PL=0
MOVL C00540 V=800.0 PL=0
MOVL C00541 V=800.0 PL=0
MOVL C00542 V=800.0 PL=0
MOVL C00543 V=800.0 PL=0
MOVL C00544 V=800.0 PL=0
MOVL C00545 V=800.0 PL=0
MOVL C00546 V=800.0 PL=0
MOVL C00547 V=800.0 PL=0
MOVL C00548 V=800.0 PL=0
MOVL C00549 V=800.0 PL=0
MOVL C00550 V=800.0 PL=0
MOVL C00551 V=800.0 PL=0
MOVL C00552 V=800.0 PL=0
MOVL C00553 V=800.0 PL=0
MOVL C00554 V=800.0 PL=0
MOVL C00555 V=800.0 PL=0
MOVL C00556 V=800.0 PL=0
MOVL C00557 V=800.0 PL=0
MOVL C00558 V=800.0 PL=0
MOVL C00559 V=800.0 PL=0
MOVL C00560 V=800.0 PL=0
MOVL C00561 V=800.0 PL=0
MOVL C00562 V=800.0 PL=0
MOVL C00563 V=800.0 PL=0
MOVL C00564 V=800.0 PL=0
MOVL C00565 V=800.0 PL=0
MOVL C00566 V=800.0 PL=0
MOVL C00567 V=800.0 PL=0
MOVL C00568 V=800.0 PL=0
MOVL C00569 V=800.0 PL=0
MOVL C00570 V=800.0 PL=0
MOVL C00571 V=800.0 PL=0
MOVL C00572 V=800.0 PL=0
MOVL C00573 V=800.0 PL=0
MOVL C00574 V=800.0 PL=0
MOVL C00575 V=800.0 PL=0
MOVL C00576 V=800.0 PL=0
MOVL C00577 V=800.0 PL=0
MOVL C00578 V=800.0 PL=0
MOVL C00579 V=800.0 PL=0
MOVL C00580 V=800.0 PL=0
MOVL C00581 V=800.0 PL=0
MOVL C00582 V=800.0 PL=0
MOVL C00583 V=800.0 PL=0
MOVL C00584 V=800.0 PL=0
MOVL C00585 V=800.0 PL=0
MOVL C00586 V=800.0 PL=0
MOVL C00587 V=800.0 PL=0
MOVL C00588 V=800.0 PL=0
MOVL C00589 V=800.0 PL=0
MOVL C00590 V=800.0 PL=0
MOVL C00591 V=800.0 PL=0
MOVL C00592 V=800.0 PL=0
MOVL C00593 V=800.0 PL=0
MOVL C00594 V=800.0 PL=0
MOVL C00595 V=800.0 PL=0
MOVL C00596 V=800.0 PL=0
MOVL C00597 V=800.0 PL=0
MOVL C00598 V=800.0 PL=0
MOVL C00599 V=800.0 PL=0
MOVL C00600 V=800.0 PL=0
MOVL C00601 V=800.0 PL=0
MOVL C00602 V=800.0 PL=0
MOVL C00603 V=800.0 PL=0
MOVL C00604 V=800.0 PL=0
MOVL C00605 V=800.0 PL=0
MOVL C00606 V=800.0 PL=0
MOVL C00607 V=800.0 PL=0
MOVL C00608 V=800.0 PL=0
MOVL C00609 V=800.0 PL=0
MOVL C00610 V=800.0 PL=0
MOVL C00611 V=800.0 PL=0
MOVL C00612 V=800.0 PL=0
MOVL C00613 V=800.0 PL=0
MOVL C00614 V=800.0 PL=0
MOVL C00615 V=800.0 PL=0
MOVL C00616 V=800.0 PL=0
MOVL C00617 V=800.0 PL=0
MOVL C00618 V=800.0 PL=0
MOVL C00619 V=800.0 PL=0
MOVL C00620 V=800.0 PL=0
MOVL C00621 V=800.0 PL=0
MOVL C00622 V=800.0 PL=0
MOVL C00623 V=800.0 PL=0
MOVL C00624 V=800.0 PL=0
MOVL C00625 V=800.0 PL=0
MOVL C00626 V=800.0 PL=0
MOVL C00627 V=800.0 PL=0
MOVL C00628 V=800.0 PL=0
MOVL C00629 V=800.0 PL=0
MOVL C00630 V=800.0 PL=0
MOVL C00631 V=800.0 PL=0
MOVL C00632 V=800.0 PL=0
MOVL C00633 V=800.0 PL=0
MOVL C00634 V=800.0 PL=0
MOVL C00635 V=800.0 PL=0
MOVL C00636 V=800.0 PL=0
MOVL C00637 V=800.0 PL=0
MOVL C00638 V=800.0 PL=0
MOVL C00639 V=800.0 PL=0
MOVL C00640 V=800.0 PL=0
MOVL C00641 V=800.0 PL=0
MOVL C00642 V=800.0 PL=0
MOVL C00643 V=800.0 PL=0
MOVL C00644 V=800.0 PL=0
MOVL C00645 V=800.0 PL=0
MOVL C00646 V=800.0 PL=0
MOVL C00647 V=800.0 PL=0
MOVL C00648 V=800.0 PL=0
MOVL C00649 V=800.0 PL=0
MOVL C00650 V=800.0 PL=0
MOVL C00651 V=800.0 PL=0
MOVL C00652 V=800.0 PL=0
MOVL C00653 V=800.0 PL=0
MOVL C00654 V=800.0 PL=0
MOVL C00655 V=800.0 PL=0
MOVL C00656 V=800.0 PL=0
MOVL C00657 V=800.0 PL=0
MOVL C00658 V=800.0 PL=0
MOVL C00659 V=800.0 PL=0
MOVL C00660 V=800.0 PL=0
MOVL C00661 V=800.0 PL=0
MOVL C00662 V=800.0 PL=0
MOVL C00663 V=800.0 PL=0
MOVL C00664 V=800.0 PL=0
MOVL C00665 V=800.0 PL=0
MOVL C00666 V=800.0 PL=0
MOVL C00667 V=800.0 PL=0
MOVL C00668 V=800.0 PL=0
MOVL C00669 V=800.0 PL=0
MOVL C00670 V=800.0 PL=0
MOVL C00671 V=800.0 PL=0
MOVL C00672 V=800.0 PL=0
MOVL C00673 V=800.0 PL=0
MOVL C00674 V=800.0 PL=0
MOVL C00675 V=800.0 PL=0
MOVL C00676 V=800.0 PL=0
MOVL C00677 V=800.0 PL=0
MOVL C00678 V=800.0 PL=0
MOVL C00679 V=800.0 PL=0
MOVL C00680 V=800.0 PL=0
MOVL C00681 V=800.0 PL=0
MOVL C00682 V=800.0 PL=0
MOVL C00683 V=800.0 PL=0
MOVL C00684 V=800.0 PL=0
MOVL C00685 V=800.0 PL=0
MOVL C00686 V=800.0 PL=0
MOVL C00687 V=800.0 PL=0
MOVL C00688 V=800.0 PL=0
MOVL C00689 V=800.0 PL=0
MOVL C00690 V=800.0 PL=0
MOVL C00691 V=800.0 PL=0
MOVL C00692 V=800.0 PL=0
MOVL C00693 V=800.0 PL=0
MOVL C00694 V=800.0 PL=0
MOVL C00695 V=800.0 PL=0
MOVL C00696 V=800.0 PL=0
MOVL C00697 V=800.0 PL=0
MOVL C00698 V=800.0 PL=0
MOVL C00699 V=800.0 PL=0
MOVL C00700 V=800.0 PL=0
MOVL C00701 V=800.0 PL=0
MOVL C00702 V=800.0 PL=0
MOVL C00703 V=800.0 PL=0
MOVL C00704 V=800.0 PL=0
MOVL C00705 V=800.0 PL=0
MOVL C00706 V=800.0 PL=0
MOVL C00707 V=800.0 PL=0
MOVL C00708 V=800.0 PL=0
MOVL C00709 V=800.0 PL=0
MOVL C00710 V=800.0 PL=0
MOVL C00711 V=800.0 PL=0
MOVL C00712 V=800.0 PL=0
MOVL C00713 V=800.0 PL=0
MOVL C00714 V=800.0 PL=0
MOVL C00715 V=800.0 PL=0
MOVL C00716 V=800.0 PL=0
MOVL C00717 V=800.0 PL=0
MOVL C00718 V=800.0 PL=0
MOVL C00719 V=800.0 PL=0
MOVL C00720 V=800.0 PL=0
MOVL C00721 V=800.0 PL=0
MOVL C00722 V=800.0 PL=0
MOVL C00723 V=800.0 PL=0
MOVL C00724 V=800.0 PL=0
MOVL C00725 V=800.0 PL=0
MOVL C00726 V=800.0 PL=0
MOVL C00727 V=800.0 PL=0
MOVL C00728 V=800.0 PL=0
MOVL C00729 V=800.0 PL=0
MOVL C00730 V=800.0 PL=0
MOVL C00731 V=800.0 PL=0
MOVL C00732 V=800.0 PL=0
MOVL C00733 V=800.0 PL=0
MOVL C00734 V=800.0 PL=0
MOVL C00735 V=800.0 PL=0
MOVL C00736 V=800.0 PL=0
MOVL C00737 V=800.0 PL=0
MOVL C00738 V=800.0 PL=0
MOVL C00739 V=800.0 PL=0
MOVL C00740 V=800.0 PL=0
MOVL C00741 V=800.0 PL=0
MOVL C00742 V=800.0 PL=0
MOVL C00743 V=800.0 PL=0
MOVL C00744 V=800.0 PL=0
MOVL C00745 V=800.0 PL=0
MOVL C00746 V=800.0 PL=0
MOVL C00747 V=800.0 PL=0
MOVL C00748 V=800.0 PL=0
MOVL C00749 V=800.0 PL=0
MOVL C00750 V=800.0 PL=0
MOVL C00751 V=800.0 PL=0
MOVL C00752 V=800.0 PL=0
MOVL C00753 V=800.0 PL=0
MOVL C00754 V=800.0 PL=0
MOVL C00755 V=800.0 PL=0
MOVL C00756 V=800.0 PL=0
MOVL C00757 V=800.0 PL=0
MOVL C00758 V=800.0 PL=0
MOVL C00759 V=800.0 PL=0
MOVL C00760 V=800.0 PL=0
MOVL C00761 V=800.0 PL=0
MOVL C00762 V=800.0 PL=0
MOVL C00763 V=800.0 PL=0
MOVL C00764 V=800.0 PL=0
MOVL C00765 V=800.0 PL=0
MOVL C00766 V=800.0 PL=0
MOVL C00767 V=800.0 PL=0
MOVL C00768 V=800.0 PL=0
MOVL C00769 V=800.0 PL=0
MOVL C00770 V=800.0 PL=0
MOVL C00771 V=800.0 PL=0
MOVL C00772 V=800.0 PL=0
MOVL C00773 V=800.0 PL=0
MOVL C00774 V=800.0 PL=0
MOVL C00775 V=800.0 PL=0
MOVL C00776 V=800.0 PL=0
MOVL C00777 V=800.0 PL=0
MOVL C00778 V=800.0 PL=0
MOVL C00779 V=800.0 PL=0
MOVL C00780 V=800.0 PL=0
MOVL C00781 V=800.0 PL=0
MOVL C00782 V=800.0 PL=0
MOVL C00783 V=800.0 PL=0
MOVL C00784 V=800.0 PL=0
MOVL C00785 V=800.0 PL=0
MOVL C00786 V=800.0 PL=0
MOVL C00787 V=800.0 PL=0
MOVL C00788 V=800.0 PL=0
MOVL C00789 V=800.0 PL=0
MOVL C00790 V=800.0 PL=0
MOVL C00791 V=800.0 PL=0
MOVL C00792 V=800.0 PL=0
MOVL C00793 V=800.0 PL=0
MOVL C00794 V=800.0 PL=0
MOVL C00795 V=800.0 PL=0
MOVL C00796 V=800.0 PL=0
MOVL C00797 V=800.0 PL=0
MOVL C00798 V=800.0 PL=0
MOVL C00799 V=800.0 PL=0
MOVL C00800 V=800.0 PL=0
MOVL C00801 V=800.0 PL=0
MOVL C00802 V=800.0 PL=0
MOVL C00803 V=800.0 PL=0
MOVL C00804 V=800.0 PL=0
MOVL C00805 V=800.0 PL=0
MOVL C00806 V=800.0 PL=0
MOVL C00807 V=800.0 PL=0
MOVL C00808 V=800.0 PL=0
MOVL C00809 V=800.0 PL=0
MOVL C00810 V=800.0 PL=0
MOVL C00811 V=800.0 PL=0
MOVL C00812 V=800.0 PL=0
MOVL C00813 V=800.0 PL=0
MOVL C00814 V=800.0 PL=0
MOVL C00815 V=800.0 PL=0
MOVL C00816 V=800.0 PL=0
MOVL C00817 V=800.0 PL=0
MOVL C00818 V=800.0 PL=0
MOVL C00819 V=800.0 PL=0
MOVL C00820 V=800.0 PL=0
MOVL C00821 V=800.0 PL=0
MOVL C00822 V=800.0 PL=0
MOVL C00823 V=800.0 PL=0
MOVL C00824 V=800.0 PL=0
MOVL C00825 V=800.0 PL=0
MOVL C00826 V=800.0 PL=0
MOVL C00827 V=800.0 PL=0
MOVL C00828 V=800.0 PL=0
MOVL C00829 V=800.0 PL=0
MOVL C00830 V=800.0 PL=0
MOVL C00831 V=800.0 PL=0
MOVL C00832 V=800.0 PL=0
MOVL C00833 V=800.0 PL=0
MOVL C00834 V=800.0 PL=0
MOVL C00835 V=800.0 PL=0
MOVL C00836 V=800.0 PL=0
MOVL C00837 V=800.0 PL=0
MOVL C00838 V=800.0 PL=0
MOVL C00839 V=800.0 PL=0
MOVL C00840 V=800.0 PL=0
MOVL C00841 V=800.0 PL=0
MOVL C00842 V=800.0 PL=0
MOVL C00843 V=800.0 PL=0
MOVL C00844 V=800.0 PL=0
MOVL C00845 V=800.0 PL=0
MOVL C00846 V=800.0 PL=0
MOVL C00847 V=800.0 PL=0
MOVL C00848 V=800.0 PL=0
MOVL C00849 V=800.0 PL=0
MOVL C00850 V=800.0 PL=0
MOVL C00851 V=800.0 PL=0
MOVL C00852 V=800.0 PL=0
MOVL C00853 V=800.0 PL=0
MOVL C00854 V=800.0 PL=0
MOVL C00855 V=800.0 PL=0
MOVL C00856 V=800.0 PL=0
MOVL C00857 V=800.0 PL=0
MOVL C00858 V=800.0 PL=0
MOVL C00859 V=800.0 PL=0
MOVL C00860 V=800.0 PL=0
MOVL C00861 V=800.0 PL=0
MOVL C00862 V=800.0 PL=0
MOVL C00863 V=800.0 PL=0
MOVL C00864 V=800.0 PL=0
MOVL C00865 V=800.0 PL=0
MOVL C00866 V=800.0 PL=0
MOVL C00867 V=800.0 PL=0
MOVL C00868 V=800.0 PL=0
MOVL C00869 V=800.0 PL=0
MOVL C00870 V=800.0 PL=0
MOVL C00871 V=800.0 PL=0
MOVL C00872 V=800.0 PL=0
MOVL C00873 V=800.0 PL=0
MOVL C00874 V=800.0 PL=0
MOVL C00875 V=800.0 PL=0
MOVL C00876 V=800.0 PL=0
MOVL C00877 V=800.0 PL=0
MOVL C00878 V=800.0 PL=0
MOVL C00879 V=800.0 PL=0
MOVL C00880 V=800.0 PL=0
MOVL C00881 V=800.0 PL=0
MOVL C00882 V=800.0 PL=0
MOVL C00883 V=800.0 PL=0
MOVL C00884 V=800.0 PL=0
MOVL C00885 V=800.0 PL=0
MOVL C00886 V=800.0 PL=0
MOVL C00887 V=800.0 PL=0
MOVL C00888 V=800.0 PL=0
MOVL C00889 V=800.0 PL=0
MOVL C00890 V=800.0 PL=0
MOVL C00891 V=800.0 PL=0
MOVL C00892 V=800.0 PL=0
MOVL C00893 V=800.0 PL=0
MOVL C00894 V=800.0 PL=0
MOVL C00895 V=800.0 PL=0
MOVL C00896 V=800.0 PL=0
MOVL C00897 V=800.0 PL=0
MOVL C00898 V=800.0 PL=0
MOVL C00899 V=800.0 PL=0
MOVL C00900 V=800.0 PL=0
MOVL C00901 V=800.0 PL=0
MOVL C00902 V=800.0 PL=0
MOVL C00903 V=800.0 PL=0
MOVL C00904 V=800.0 PL=0
MOVL C00905 V=800.0 PL=0
MOVL C00906 V=800.0 PL=0
MOVL C00907 V=800.0 PL=0
MOVL C00908 V=800.0 PL=0
MOVL C00909 V=800.0 PL=0
MOVL C00910 V=800.0 PL=0
MOVL C00911 V=800.0 PL=0
MOVL C00912 V=800.0 PL=0
MOVL C00913 V=800.0 PL=0
MOVL C00914 V=800.0 PL=0
MOVL C00915 V=800.0 PL=0
MOVL C00916 V=800.0 PL=0
MOVL C00917 V=800.0 PL=0
MOVL C00918 V=800.0 PL=0
MOVL C00919 V=800.0 PL=0
MOVL C00920 V=800.0 PL=0
MOVL C00921 V=800.0 PL=0
MOVL C00922 V=800.0 PL=0
MOVL C00923 V=800.0 PL=0
MOVL C00924 V=800.0 PL=0
MOVL C00925 V=800.0 PL=0
MOVL C00926 V=800.0 PL=0
MOVL C00927 V=800.0 PL=0
MOVL C00928 V=800.0 PL=0
MOVL C00929 V=800.0 PL=0
MOVL C00930 V=800.0 PL=0
MOVL C00931 V=800.0 PL=0
MOVL C00932 V=800.0 PL=0
MOVL C00933 V=800.0 PL=0
MOVL C00934 V=800.0 PL=0
MOVL C00935 V=800.0 PL=0
MOVL C00936 V=800.0 PL=0
MOVL C00937 V=800.0 PL=0
MOVL C00938 V=800.0 PL=0
MOVL C00939 V=800.0 PL=0
MOVL C00940 V=800.0 PL=0
MOVL C00941 V=800.0 PL=0
MOVL C00942 V=800.0 PL=0
MOVL C00943 V=800.0 PL=0
MOVL C00944 V=800.0 PL=0
MOVL C00945 V=800.0 PL=0
MOVL C00946 V=800.0 PL=0
MOVL C00947 V=800.0 PL=0
MOVL C00948 V=800.0 PL=0
MOVL C00949 V=800.0 PL=0
MOVL C00950 V=800.0 PL=0
MOVL C00951 V=800.0 PL=0
MOVL C00952 V=800.0 PL=0
MOVL C00953 V=800.0 PL=0
MOVL C00954 V=800.0 PL=0
MOVL C00955 V=800.0 PL=0
MOVL C00956 V=800.0 PL=0
MOVL C00957 V=800.0 PL=0
MOVL C00958 V=800.0 PL=0
MOVL C00959 V=800.0 PL=0
MOVL C00960 V=800.0 PL=0
MOVL C00961 V=800.0 PL=0
MOVL C00962 V=800.0 PL=0
MOVL C00963 V=800.0 PL=0
MOVL C00964 V=800.0 PL=0
MOVL C00965 V=800.0 PL=0
MOVL C00966 V=800.0 PL=0
MOVL C00967 V=800.0 PL=0
MOVL C00968 V=800.0 PL=0
MOVL C00969 V=800.0 PL=0
MOVL C00970 V=800.0 PL=0
MOVL C00971 V=800.0 PL=0
MOVL C00972 V=800.0 PL=0
MOVL C00973 V=800.0 PL=0
MOVL C00974 V=800.0 PL=0
MOVL C00975 V=800.0 PL=0
MOVL C00976 V=800.0 PL=0
MOVL C00977 V=800.0 PL=0
MOVL C00978 V=800.0 PL=0
MOVL C00979 V=800.0 PL=0
MOVL C00980 V=800.0 PL=0
MOVL C00981 V=800.0 PL=0
MOVL C00982 V=800.0 PL=0
MOVL C00983 V=800.0 PL=0
MOVL C00984 V=800.0 PL=0
MOVL C00985 V=800.0 PL=0
MOVL C00986 V=800.0 PL=0
MOVL C00987 V=800.0 PL=0
MOVL C00988 V=800.0 PL=0
MOVL C00989 V=800.0 PL=0
MOVL C00990 V=800.0 PL=0
MOVL C00991 V=800.0 PL=0
MOVL C00992 V=800.0 PL=0
MOVL C00993 V=800.0 PL=0
MOVL C00994 V=800.0 PL=0
MOVL C00995 V=800.0 PL=0
MOVL C00996 V=800.0 PL=0
MOVL C00997 V=800.0 PL=0
MOVL C00998 V=800.0 PL=0
MOVL C00999 V=800.0 PL=0
MOVL C01000 V=800.0 PL=0
MOVL C01001 V=800.0 PL=0
MOVL C01002 V=800.0 PL=0
MOVL C01003 V=800.0 PL=0
MOVL C01004 V=800.0 PL=0
MOVL C01005 V=800.0 PL=0
MOVL C01006 V=800.0 PL=0
MOVL C01007 V=800.0 PL=0
MOVL C01008 V=800.0 PL=0
MOVL C01009 V=800.0 PL=0
MOVL C01010 V=800.0 PL=0
MOVL C01011 V=800.0 PL=0
MOVL C01012 V=800.0 PL=0
MOVL C01013 V=800.0 PL=0
MOVL C01014 V=800.0 PL=0
MOVL C01015 V=800.0 PL=0
MOVL C01016 V=800.0 PL=0
MOVL C01017 V=800.0 PL=0
MOVL C01018 V=800.0 PL=0
MOVL C01019 V=800.0 PL=0
MOVL C01020 V=800.0 PL=0
MOVL C01021 V=800.0 PL=0
MOVL C01022 V=800.0 PL=0
MOVL C01023 V=800.0 PL=0
MOVL C01024 V=800.0 PL=0
MOVL C01025 V=800.0 PL=0
MOVL C01026 V=800.0 PL=0
MOVL C01027 V=800.0 PL=0
MOVL C01028 V=800.0 PL=0
MOVL C01029 V=800.0 PL=0
MOVL C01030 V=800.0 PL=0
MOVL C01031 V=800.0 PL=0
MOVL C01032 V=800.0 PL=0
MOVL C01033 V=800.0 PL=0
MOVL C01034 V=800.0 PL=0
MOVL C01035 V=800.0 PL=0
MOVL C01036 V=800.0 PL=0
MOVL C01037 V=800.0 PL=0
MOVL C01038 V=800.0 PL=0
MOVL C01039 V=800.0 PL=0
MOVL C01040 V=800.0 PL=0
MOVL C01041 V=800.0 PL=0
MOVL C01042 V=800.0 PL=0
MOVL C01043 V=800.0 PL=0
MOVL C01044 V=800.0 PL=0
MOVL C01045 V=800.0 PL=0
MOVL C01046 V=800.0 PL=0
MOVL C01047 V=800.0 PL=0
MOVL C01048 V=800.0 PL=0
MOVL C01049 V=800.0 PL=0
MOVL C01050 V=800.0 PL=0
MOVL C01051 V=800.0 PL=0
MOVL C01052 V=800.0 PL=0
MOVL C01053 V=800.0 PL=0
MOVL C01054 V=800.0 PL=0
MOVL C01055 V=800.0 PL=0
MOVL C01056 V=800.0 PL=0
MOVL C01057 V=800.0 PL=0
MOVL C01058 V=800.0 PL=0
MOVL C01059 V=800.0 PL=0
MOVL C01060 V=800.0 PL=0
MOVL C01061 V=800.0 PL=0
MOVL C01062 V=800.0 PL=0
MOVL C01063 V=800.0 PL=0
MOVL C01064 V=800.0 PL=0
MOVL C01065 V=800.0 PL=0
MOVL C01066 V=800.0 PL=0
MOVL C01067 V=800.0 PL=0
MOVL C01068 V=800.0 PL=0
MOVL C01069 V=800.0 PL=0
MOVL C01070 V=800.0 PL=0
MOVL C01071 V=800.0 PL=0
MOVL C01072 V=800.0 PL=0
MOVL C01073 V=800.0 PL=0
MOVL C01074 V=800.0 PL=0
MOVL C01075 V=800.0 PL=0
MOVL C01076 V=800.0 PL=0
MOVL C01077 V=800.0 PL=0
MOVL C01078 V=800.0 PL=0
MOVL C01079 V=800.0 PL=0
MOVL C01080 V=800.0 PL=0
MOVL C01081 V=800.0 PL=0
MOVL C01082 V=800.0 PL=0
MOVL C01083 V=800.0 PL=0
MOVL C01084 V=800.0 PL=0
MOVL C01085 V=800.0 PL=0
MOVL C01086 V=800.0 PL=0
MOVL C01087 V=800.0 PL=0
MOVL C01088 V=800.0 PL=0
MOVL C01089 V=800.0 PL=0
MOVL C01090 V=800.0 PL=0
MOVL C01091 V=800.0 PL=0
MOVL C01092 V=800.0 PL=0
MOVL C01093 V=800.0 PL=0
MOVL C01094 V=800.0 PL=0
MOVL C01095 V=800.0 PL=0
MOVL C01096 V=800.0 PL=0
MOVL C01097 V=800.0 PL=0
MOVL C01098 V=800.0 PL=0
MOVL C01099 V=800.0 PL=0
MOVL C01100 V=800.0 PL=0
MOVL C01101 V=800.0 PL=0
MOVL C01102 V=800.0 PL=0
MOVL C01103 V=800.0 PL=0
MOVL C01104 V=800.0 PL=0
MOVL C01105 V=800.0 PL=0
MOVL C01106 V=800.0 PL=0
MOVL C01107 V=800.0 PL=0
MOVL C01108 V=800.0 PL=0
MOVL C01109 V=800.0 PL=0
MOVL C01110 V=800.0 PL=0
MOVL C01111 V=800.0 PL=0
MOVL C01112 V=800.0 PL=0
MOVL C01113 V=800.0 PL=0
MOVL C01114 V=800.0 PL=0
MOVL C01115 V=800.0 PL=0
MOVL C01116 V=800.0 PL=0
MOVL C01117 V=800.0 PL=0
MOVL C01118 V=800.0 PL=0
MOVL C01119 V=800.0 PL=0
MOVL C01120 V=800.0 PL=0
MOVL C01121 V=800.0 PL=0
MOVL C01122 V=800.0 PL=0
MOVL C01123 V=800.0 PL=0
MOVL C01124 V=800.0 PL=0
MOVL C01125 V=800.0 PL=0
MOVL C01126 V=800.0 PL=0
MOVL C01127 V=800.0 PL=0
MOVL C01128 V=800.0 PL=0
MOVL C01129 V=800.0 PL=0
MOVL C01130 V=800.0 PL=0
MOVL C01131 V=800.0 PL=0
MOVL C01132 V=800.0 PL=0
MOVL C01133 V=800.0 PL=0
MOVL C01134 V=800.0 PL=0
MOVL C01135 V=800.0 PL=0
MOVL C01136 V=800.0 PL=0
MOVL C01137 V=800.0 PL=0
MOVL C01138 V=800.0 PL=0
MOVL C01139 V=800.0 PL=0
MOVL C01140 V=800.0 PL=0
MOVL C01141 V=800.0 PL=0
MOVL C01142 V=800.0 PL=0
MOVL C01143 V=800.0 PL=0
MOVL C01144 V=800.0 PL=0
MOVL C01145 V=800.0 PL=0
MOVL C01146 V=800.0 PL=0
MOVL C01147 V=800.0 PL=0
MOVL C01148 V=800.0 PL=0
MOVL C01149 V=800.0 PL=0
MOVL C01150 V=800.0 PL=0
MOVL C01151 V=800.0 PL=0
MOVL C01152 V=800.0 PL=0
MOVL C01153 V=800.0 PL=0
MOVL C01154 V=800.0 PL=0
MOVL C01155 V=800.0 PL=0
MOVL C01156 V=800.0 PL=0
MOVL C01157 V=800.0 PL=0
MOVL C01158 V=800.0 PL=0
MOVL C01159 V=800.0 PL=0
MOVL C01160 V=800.0 PL=0
MOVL C01161 V=800.0 PL=0
MOVL C01162 V=800.0 PL=0
MOVL C01163 V=800.0 PL=0
MOVL C01164 V=800.0 PL=0
MOVL C01165 V=800.0 PL=0
MOVL C01166 V=800.0 PL=0
MOVL C01167 V=800.0 PL=0
MOVL C01168 V=800.0 PL=0
MOVL C01169 V=800.0 PL=0
MOVL C01170 V=800.0 PL=0
MOVL C01171 V=800.0 PL=0
MOVL C01172 V=800.0 PL=0
MOVL C01173 V=800.0 PL=0
MOVL C01174 V=800.0 PL=0
MOVL C01175 V=800.0 PL=0
MOVL C01176 V=800.0 PL=0
MOVL C01177 V=800.0 PL=0
MOVL C01178 V=800.0 PL=0
MOVL C01179 V=800.0 PL=0
MOVL C01180 V=800.0 PL=0
MOVL C01181 V=800.0 PL=0
MOVL C01182 V=800.0 PL=0
MOVL C01183 V=800.0 PL=0
MOVL C01184 V=800.0 PL=0
MOVL C01185 V=800.0 PL=0
MOVL C01186 V=800.0 PL=0
MOVL C01187 V=800.0 PL=0
MOVL C01188 V=800.0 PL=0
MOVL C01189 V=800.0 PL=0
MOVL C01190 V=800.0 PL=0
MOVL C01191 V=800.0 PL=0
MOVL C01192 V=800.0 PL=0
MOVL C01193 V=800.0 PL=0
MOVL C01194 V=800.0 PL=0
MOVL C01195 V=800.0 PL=0
MOVL C01196 V=800.0 PL=0
MOVL C01197 V=800.0 PL=0
MOVL C01198 V=800.0 PL=0
MOVL C01199 V=800.0 PL=0
MOVL C01200 V=800.0 PL=0
MOVL C01201 V=800.0 PL=0
MOVL C01202 V=800.0 PL=0
MOVL C01203 V=800.0 PL=0
MOVL C01204 V=800.0 PL=0
MOVL C01205 V=800.0 PL=0
MOVL C01206 V=800.0 PL=0
MOVL C01207 V=800.0 PL=0
MOVL C01208 V=800.0 PL=0
MOVL C01209 V=800.0 PL=0
MOVL C01210 V=800.0 PL=0
MOVL C01211 V=800.0 PL=0
MOVL C01212 V=800.0 PL=0
MOVL C01213 V=800.0 PL=0
MOVL C01214 V=800.0 PL=0
MOVL C01215 V=800.0 PL=0
MOVL C01216 V=800.0 PL=0
MOVL C01217 V=800.0 PL=0
MOVL C01218 V=800.0 PL=0
MOVL C01219 V=800.0 PL=0
MOVL C01220 V=800.0 PL=0
MOVL C01221 V=800.0 PL=0
MOVL C01222 V=800.0 PL=0
MOVL C01223 V=800.0 PL=0
MOVL C01224 V=800.0 PL=0
MOVL C01225 V=800.0 PL=0
MOVL C01226 V=800.0 PL=0
MOVL C01227 V=800.0 PL=0
MOVL C01228 V=800.0 PL=0
MOVL C01229 V=800.0 PL=0
MOVL C01230 V=800.0 PL=0
MOVL C01231 V=800.0 PL=0
MOVL C01232 V=800.0 PL=0
MOVL C01233 V=800.0 PL=0
MOVL C01234 V=800.0 PL=0
MOVL C01235 V=800.0 PL=0
MOVL C01236 V=800.0 PL=0
MOVL C01237 V=800.0 PL=0
MOVL C01238 V=800.0 PL=0
MOVL C01239 V=800.0 PL=0
MOVL C01240 V=800.0 PL=0
MOVL C01241 V=800.0 PL=0
MOVL C01242 V=800.0 PL=0
MOVL C01243 V=800.0 PL=0
MOVL C01244 V=800.0 PL=0
MOVL C01245 V=800.0 PL=0
MOVL C01246 V=800.0 PL=0
MOVL C01247 V=800.0 PL=0
MOVL C01248 V=800.0 PL=0
MOVL C01249 V=800.0 PL=0
MOVL C01250 V=800.0 PL=0
MOVL C01251 V=800.0 PL=0
MOVL C01252 V=800.0 PL=0
MOVL C01253 V=800.0 PL=0
MOVL C01254 V=800.0 PL=0
MOVL C01255 V=800.0 PL=0
MOVL C01256 V=800.0 PL=0
MOVL C01257 V=800.0 PL=0
MOVL C01258 V=800.0 PL=0
MOVL C01259 V=800.0 PL=0
MOVL C01260 V=800.0 PL=0
MOVL C01261 V=800.0 PL=0
MOVL C01262 V=800.0 PL=0
MOVL C01263 V=800.0 PL=0
MOVL C01264 V=800.0 PL=0
MOVL C01265 V=800.0 PL=0
MOVL C01266 V=800.0 PL=0
MOVL C01267 V=800.0 PL=0
MOVL C01268 V=800.0 PL=0
MOVL C01269 V=800.0 PL=0
MOVL C01270 V=800.0 PL=0
MOVL C01271 V=800.0 PL=0
MOVL C01272 V=800.0 PL=0
MOVL C01273 V=800.0 PL=0
MOVL C01274 V=800.0 PL=0
MOVL C01275 V=800.0 PL=0
MOVL C01276 V=800.0 PL=0
MOVL C01277 V=800.0 PL=0
MOVL C01278 V=800.0 PL=0
MOVL C01279 V=800.0 PL=0
MOVL C01280 V=800.0 PL=0
MOVL C01281 V=800.0 PL=0
MOVL C01282 V=800.0 PL=0
MOVL C01283 V=800.0 PL=0
MOVL C01284 V=800.0 PL=0
MOVL C01285 V=800.0 PL=0
MOVL C01286 V=800.0 PL=0
MOVL C01287 V=800.0 PL=0
MOVL C01288 V=800.0 PL=0
MOVL C01289 V=800.0 PL=0
MOVL C01290 V=800.0 PL=0
MOVL C01291 V=800.0 PL=0
MOVL C01292 V=800.0 PL=0
MOVL C01293 V=800.0 PL=0
MOVL C01294 V=800.0 PL=0
MOVL C01295 V=800.0 PL=0
MOVL C01296 V=800.0 PL=0
MOVL C01297 V=800.0 PL=0
MOVL C01298 V=800.0 PL=0
MOVL C01299 V=800.0 PL=0
MOVL C01300 V=800.0 PL=0
MOVL C01301 V=800.0 PL=0
MOVL C01302 V=800.0 PL=0
MOVL C01303 V=800.0 PL=0
MOVL C01304 V=800.0 PL=0
MOVL C01305 V=800.0 PL=0
MOVL C01306 V=800.0 PL=0
MOVL C01307 V=800.0 PL=0
MOVL C01308 V=800.0 PL=0
MOVL C01309 V=800.0 PL=0
MOVL C01310 V=800.0 PL=0
MOVL C01311 V=800.0 PL=0
MOVL C01312 V=800.0 PL=0
MOVL C01313 V=800.0 PL=0
MOVL C01314 V=800.0 PL=0
MOVL C01315 V=800.0 PL=0
MOVL C01316 V=800.0 PL=0
MOVL C01317 V=800.0 PL=0
MOVL C01318 V=800.0 PL=0
MOVL C01319 V=800.0 PL=0
MOVL C01320 V=800.0 PL=0
MOVL C01321 V=800.0 PL=0
MOVL C01322 V=800.0 PL=0
MOVL C01323 V=800.0 PL=0
MOVL C01324 V=800.0 PL=0
MOVL C01325 V=800.0 PL=0
MOVL C01326 V=800.0 PL=0
MOVL C01327 V=800.0 PL=0
MOVL C01328 V=800.0 PL=0
MOVL C01329 V=800.0 PL=0
MOVL C01330 V=800.0 PL=0
MOVL C01331 V=800.0 PL=0
MOVL C01332 V=800.0 PL=0
MOVL C01333 V=800.0 PL=0
MOVL C01334 V=800.0 PL=0
MOVL C01335 V=800.0 PL=0
MOVL C01336 V=800.0 PL=0
MOVL C01337 V=800.0 PL=0
MOVL C01338 V=800.0 PL=0
MOVL C01339 V=800.0 PL=0
MOVL C01340 V=800.0 PL=0
MOVL C01341 V=800.0 PL=0
MOVL C01342 V=800.0 PL=0
MOVL C01343 V=800.0 PL=0
MOVL C01344 V=800.0 PL=0
MOVL C01345 V=800.0 PL=0
MOVL C01346 V=800.0 PL=0
MOVL C01347 V=800.0 PL=0
MOVL C01348 V=800.0 PL=0
MOVL C01349 V=800.0 PL=0
MOVL C01350 V=800.0 PL=0
MOVL C01351 V=800.0 PL=0
MOVL C01352 V=800.0 PL=0
MOVL C01353 V=800.0 PL=0
MOVL C01354 V=800.0 PL=0
MOVL C01355 V=800.0 PL=0
MOVL C01356 V=800.0 PL=0
MOVL C01357 V=800.0 PL=0
MOVL C01358 V=800.0 PL=0
MOVL C01359 V=800.0 PL=0
MOVL C01360 V=800.0 PL=0
MOVL C01361 V=800.0 PL=0
MOVL C01362 V=800.0 PL=0
MOVL C01363 V=800.0 PL=0
MOVL C01364 V=800.0 PL=0
MOVL C01365 V=800.0 PL=0
MOVL C01366 V=800.0 PL=0
MOVL C01367 V=800.0 PL=0
MOVL C01368 V=800.0 PL=0
MOVL C01369 V=800.0 PL=0
MOVL C01370 V=800.0 PL=0
MOVL C01371 V=800.0 PL=0
MOVL C01372 V=800.0 PL=0
MOVL C01373 V=800.0 PL=0
MOVL C01374 V=800.0 PL=0
MOVL C01375 V=800.0 PL=0
MOVL C01376 V=800.0 PL=0
MOVL C01377 V=800.0 PL=0
MOVL C01378 V=800.0 PL=0
MOVL C01379 V=800.0 PL=0
MOVL C01380 V=800.0 PL=0
MOVL C01381 V=800.0 PL=0
MOVL C01382 V=800.0 PL=0
MOVL C01383 V=800.0 PL=0
MOVL C01384 V=800.0 PL=0
MOVL C01385 V=800.0 PL=0
MOVL C01386 V=800.0 PL=0
MOVL C01387 V=800.0 PL=0
MOVL C01388 V=800.0 PL=0
MOVL C01389 V=800.0 PL=0
MOVL C01390 V=800.0 PL=0
MOVL C01391 V=800.0 PL=0
MOVL C01392 V=800.0 PL=0
MOVL C01393 V=800.0 PL=0
MOVL C01394 V=800.0 PL=0
MOVL C01395 V=800.0 PL=0
MOVL C01396 V=800.0 PL=0
MOVL C01397 V=800.0 PL=0
MOVL C01398 V=800.0 PL=0
MOVL C01399 V=800.0 PL=0
MOVL C01400 V=800.0 PL=0
MOVL C01401 V=800.0 PL=0
MOVL C01402 V=800.0 PL=0
MOVL C01403 V=800.0 PL=0
MOVL C01404 V=800.0 PL=0
MOVL C01405 V=800.0 PL=0
MOVL C01406 V=800.0 PL=0
MOVL C01407 V=800.0 PL=0
MOVL C01408 V=800.0 PL=0
MOVL C01409 V=800.0 PL=0
MOVL C01410 V=800.0 PL=0
MOVL C01411 V=800.0 PL=0
MOVL C01412 V=800.0 PL=0
MOVL C01413 V=800.0 PL=0
MOVL C01414 V=800.0 PL=0
MOVL C01415 V=800.0 PL=0
MOVL C01416 V=800.0 PL=0
MOVL C01417 V=800.0 PL=0
MOVL C01418 V=800.0 PL=0
MOVL C01419 V=800.0 PL=0
MOVL C01420 V=800.0 PL=0
MOVL C01421 V=800.0 PL=0
MOVL C01422 V=800.0 PL=0
MOVL C01423 V=800.0 PL=0
MOVL C01424 V=800.0 PL=0
MOVL C01425 V=800.0 PL=0
MOVL C01426 V=800.0 PL=0
MOVL C01427 V=800.0 PL=0
MOVL C01428 V=800.0 PL=0
MOVL C01429 V=800.0 PL=0
MOVL C01430 V=800.0 PL=0
MOVL C01431 V=800.0 PL=0
MOVL C01432 V=800.0 PL=0
MOVL C01433 V=800.0 PL=0
MOVL C01434 V=800.0 PL=0
MOVL C01435 V=800.0 PL=0
MOVL C01436 V=800.0 PL=0
MOVL C01437 V=800.0 PL=0
MOVL C01438 V=800.0 PL=0
MOVL C01439 V=800.0 PL=0
MOVL C01440 V=800.0 PL=0
MOVL C01441 V=800.0 PL=0
MOVL C01442 V=800.0 PL=0
MOVL C01443 V=800.0 PL=0
MOVL C01444 V=800.0 PL=0
MOVL C01445 V=800.0 PL=0
MOVL C01446 V=800.0 PL=0
MOVL C01447 V=800.0 PL=0
MOVL C01448 V=800.0 PL=0
MOVL C01449 V=800.0 PL=0
MOVL C01450 V=800.0 PL=0
MOVL C01451 V=800.0 PL=0
MOVL C01452 V=800.0 PL=0
MOVL C01453 V=800.0 PL=0
MOVL C01454 V=800.0 PL=0
MOVL C01455 V=800.0 PL=0
MOVL C01456 V=800.0 PL=0
MOVL C01457 V=800.0 PL=0
MOVL C01458 V=800.0 PL=0
MOVL C01459 V=800.0 PL=0
MOVL C01460 V=800.0 PL=0
MOVL C01461 V=800.0 PL=0
MOVL C01462 V=800.0 PL=0
MOVL C01463 V=800.0 PL=0
MOVL C01464 V=800.0 PL=0
MOVL C01465 V=800.0 PL=0
MOVL C01466 V=800.0 PL=0
MOVL C01467 V=800.0 PL=0
MOVL C01468 V=800.0 PL=0
MOVL C01469 V=800.0 PL=0
MOVL C01470 V=800.0 PL=0
MOVL C01471 V=800.0 PL=0
MOVL C01472 V=800.0 PL=0
MOVL C01473 V=800.0 PL=0
MOVL C01474 V=800.0 PL=0
MOVL C01475 V=800.0 PL=0
MOVL C01476 V=800.0 PL=0
MOVL C01477 V=800.0 PL=0
MOVL C01478 V=800.0 PL=0
MOVL C01479 V=800.0 PL=0
MOVL C01480 V=800.0 PL=0
MOVL C01481 V=800.0 PL=0
MOVL C01482 V=800.0 PL=0
MOVL C01483 V=800.0 PL=0
MOVL C01484 V=800.0 PL=0
MOVL C01485 V=800.0 PL=0
MOVL C01486 V=800.0 PL=0
MOVL C01487 V=800.0 PL=0
MOVL C01488 V=800.0 PL=0
MOVL C01489 V=800.0 PL=0
MOVL C01490 V=800.0 PL=0
MOVL C01491 V=800.0 PL=0
MOVL C01492 V=800.0 PL=0
MOVL C01493 V=800.0 PL=0
MOVL C01494 V=800.0 PL=0
MOVL C01495 V=800.0 PL=0
MOVL C01496 V=800.0 PL=0
MOVL C01497 V=800.0 PL=0
MOVL C01498 V=800.0 PL=0
MOVL C01499 V=800.0 PL=0
MOVL C01500 V=800.0 PL=0
MOVL C01501 V=800.0 PL=0
MOVL C01502 V=800.0 PL=0
MOVL C01503 V=800.0 PL=0
MOVL C01504 V=800.0 PL=0
MOVL C01505 V=800.0 PL=0
MOVL C01506 V=800.0 PL=0
MOVL C01507 V=800.0 PL=0
MOVL C01508 V=800.0 PL=0
MOVL C01509 V=800.0 PL=0
MOVL C01510 V=800.0 PL=0
MOVL C01511 V=800.0 PL=0
MOVL C01512 V=800.0 PL=0
MOVL C01513 V=800.0 PL=0
MOVL C01514 V=800.0 PL=0
MOVL C01515 V=800.0 PL=0
MOVL C01516 V=800.0 PL=0
MOVL C01517 V=800.0 PL=0
MOVL C01518 V=800.0 PL=0
MOVL C01519 V=800.0 PL=0
MOVL C01520 V=800.0 PL=0
MOVL C01521 V=800.0 PL=0
MOVL C01522 V=800.0 PL=0
MOVL C01523 V=800.0 PL=0
MOVL C01524 V=800.0 PL=0
MOVL C01525 V=800.0 PL=0
MOVL C01526 V=800.0 PL=0
MOVL C01527 V=800.0 PL=0
MOVL C01528 V=800.0 PL=0
MOVL C01529 V=800.0 PL=0
MOVL C01530 V=800.0 PL=0
MOVL C01531 V=800.0 PL=0
MOVL C01532 V=800.0 PL=0
MOVL C01533 V=800.0 PL=0
MOVL C01534 V=800.0 PL=0
MOVL C01535 V=800.0 PL=0
MOVL C01536 V=800.0 PL=0
MOVL C01537 V=800.0 PL=0
MOVL C01538 V=800.0 PL=0
MOVL C01539 V=800.0 PL=0
MOVL C01540 V=800.0 PL=0
MOVL C01541 V=800.0 PL=0
MOVL C01542 V=800.0 PL=0
MOVL C01543 V=800.0 PL=0
MOVL C01544 V=800.0 PL=0
MOVL C01545 V=800.0 PL=0
MOVL C01546 V=800.0 PL=0
MOVL C01547 V=800.0 PL=0
MOVL C01548 V=800.0 PL=0
MOVL C01549 V=800.0 PL=0
MOVL C01550 V=800.0 PL=0
MOVL C01551 V=800.0 PL=0
MOVL C01552 V=800.0 PL=0
MOVL C01553 V=800.0 PL=0
MOVL C01554 V=800.0 PL=0
MOVL C01555 V=800.0 PL=0
MOVL C01556 V=800.0 PL=0
MOVL C01557 V=800.0 PL=0
MOVL C01558 V=800.0 PL=0
MOVL C01559 V=800.0 PL=0
MOVL C01560 V=800.0 PL=0
MOVL C01561 V=800.0 PL=0
MOVL C01562 V=800.0 PL=0
MOVL C01563 V=800.0 PL=0
MOVL C01564 V=800.0 PL=0
MOVL C01565 V=800.0 PL=0
MOVL C01566 V=800.0 PL=0
MOVL C01567 V=800.0 PL=0
MOVL C01568 V=800.0 PL=0
MOVL C01569 V=800.0 PL=0
MOVL C01570 V=800.0 PL=0
MOVL C01571 V=800.0 PL=0
MOVL C01572 V=800.0 PL=0
MOVL C01573 V=800.0 PL=0
MOVL C01574 V=800.0 PL=0
MOVL C01575 V=800.0 PL=0
MOVL C01576 V=800.0 PL=0
MOVL C01577 V=800.0 PL=0
MOVL C01578 V=800.0 PL=0
MOVL C01579 V=800.0 PL=0
MOVL C01580 V=800.0 PL=0
MOVL C01581 V=800.0 PL=0
MOVL C01582 V=800.0 PL=0
MOVL C01583 V=800.0 PL=0
MOVL C01584 V=800.0 PL=0
MOVL C01585 V=800.0 PL=0
MOVL C01586 V=800.0 PL=0
MOVL C01587 V=800.0 PL=0
MOVL C01588 V=800.0 PL=0
MOVL C01589 V=800.0 PL=0
MOVL C01590 V=800.0 PL=0
MOVL C01591 V=800.0 PL=0
MOVL C01592 V=800.0 PL=0
MOVL C01593 V=800.0 PL=0
MOVL C01594 V=800.0 PL=0
MOVL C01595 V=800.0 PL=0
MOVL C01596 V=800.0 PL=0
MOVL C01597 V=800.0 PL=0
MOVL C01598 V=800.0 PL=0
MOVL C01599 V=800.0 PL=0
MOVL C01600 V=800.0 PL=0
MOVL C01601 V=800.0 PL=0
MOVL C01602 V=800.0 PL=0
MOVL C01603 V=800.0 PL=0
MOVL C01604 V=800.0 PL=0
MOVL C01605 V=800.0 PL=0
MOVL C01606 V=800.0 PL=0
MOVL C01607 V=800.0 PL=0
MOVL C01608 V=800.0 PL=0
MOVL C01609 V=800.0 PL=0
MOVL C01610 V=800.0 PL=0
MOVL C01611 V=800.0 PL=0
MOVL C01612 V=800.0 PL=0
MOVL C01613 V=800.0 PL=0
MOVL C01614 V=800.0 PL=0
MOVL C01615 V=800.0 PL=0
MOVL C01616 V=800.0 PL=0
MOVL C01617 V=800.0 PL=0
MOVL C01618 V=800.0 PL=0
MOVL C01619 V=800.0 PL=0
MOVL C01620 V=800.0 PL=0
MOVL C01621 V=800.0 PL=0
MOVL C01622 V=800.0 PL=0
MOVL C01623 V=800.0 PL=0
MOVL C01624 V=800.0 PL=0
MOVL C01625 V=800.0 PL=0
MOVL C01626 V=800.0 PL=0
MOVL C01627 V=800.0 PL=0
MOVL C01628 V=800.0 PL=0
MOVL C01629 V=800.0 PL=0
MOVL C01630 V=800.0 PL=0
MOVL C01631 V=800.0 PL=0
MOVL C01632 V=800.0 PL=0
MOVL C01633 V=800.0 PL=0
MOVL C01634 V=800.0 PL=0
MOVL C01635 V=800.0 PL=0
MOVL C01636 V=800.0 PL=0
MOVL C01637 V=800.0 PL=0
MOVL C01638 V=800.0 PL=0
MOVL C01639 V=800.0 PL=0
MOVL C01640 V=800.0 PL=0
MOVL C01641 V=800.0 PL=0
MOVL C01642 V=800.0 PL=0
MOVL C01643 V=800.0 PL=0
MOVL C01644 V=800.0 PL=0
MOVL C01645 V=800.0 PL=0
MOVL C01646 V=800.0 PL=0
MOVL C01647 V=800.0 PL=0
MOVL C01648 V=800.0 PL=0
MOVL C01649 V=800.0 PL=0
MOVL C01650 V=800.0 PL=0
MOVL C01651 V=800.0 PL=0
MOVL C01652 V=800.0 PL=0
MOVL C01653 V=800.0 PL=0
MOVL C01654 V=800.0 PL=0
MOVL C01655 V=800.0 PL=0
MOVL C01656 V=800.0 PL=0
MOVL C01657 V=800.0 PL=0
MOVL C01658 V=800.0 PL=0
MOVL C01659 V=800.0 PL=0
MOVL C01660 V=800.0 PL=0
MOVL C01661 V=800.0 PL=0
MOVL C01662 V=800.0 PL=0
MOVL C01663 V=800.0 PL=0
MOVL C01664 V=800.0 PL=0
MOVL C01665 V=800.0 PL=0
MOVL C01666 V=800.0 PL=0
MOVL C01667 V=800.0 PL=0
MOVL C01668 V=800.0 PL=0
MOVL C01669 V=800.0 PL=0
MOVL C01670 V=800.0 PL=0
MOVL C01671 V=800.0 PL=0
MOVL C01672 V=800.0 PL=0
MOVL C01673 V=800.0 PL=0
MOVL C01674 V=800.0 PL=0
MOVL C01675 V=800.0 PL=0
MOVL C01676 V=800.0 PL=0
MOVL C01677 V=800.0 PL=0
MOVL C01678 V=800.0 PL=0
MOVL C01679 V=800.0 PL=0
MOVL C01680 V=800.0 PL=0
MOVL C01681 V=800.0 PL=0
MOVL C01682 V=800.0 PL=0
MOVL C01683 V=800.0 PL=0
MOVL C01684 V=800.0 PL=0
MOVL C01685 V=800.0 PL=0
MOVL C01686 V=800.0 PL=0
MOVL C01687 V=800.0 PL=0
MOVL C01688 V=800.0 PL=0
MOVL C01689 V=800.0 PL=0
MOVL C01690 V=800.0 PL=0
MOVL C01691 V=800.0 PL=0
MOVL C01692 V=800.0 PL=0
MOVL C01693 V=800.0 PL=0
MOVL C01694 V=800.0 PL=0
MOVL C01695 V=800.0 PL=0
MOVL C01696 V=800.0 PL=0
MOVL C01697 V=800.0 PL=0
MOVL C01698 V=800.0 PL=0
MOVL C01699 V=800.0 PL=0
MOVL C01700 V=800.0 PL=0
MOVL C01701 V=800.0 PL=0
MOVL C01702 V=800.0 PL=0
MOVL C01703 V=800.0 PL=0
MOVL C01704 V=800.0 PL=0
MOVL C01705 V=800.0 PL=0
MOVL C01706 V=800.0 PL=0
MOVL C01707 V=800.0 PL=0
MOVL C01708 V=800.0 PL=0
MOVL C01709 V=800.0 PL=0
MOVL C01710 V=800.0 PL=0
MOVL C01711 V=800.0 PL=0
MOVL C01712 V=800.0 PL=0
MOVL C01713 V=800.0 PL=0
MOVL C01714 V=800.0 PL=0
MOVL C01715 V=800.0 PL=0
MOVL C01716 V=800.0 PL=0
MOVL C01717 V=800.0 PL=0
MOVL C01718 V=800.0 PL=0
MOVL C01719 V=800.0 PL=0
MOVL C01720 V=800.0 PL=0
MOVL C01721 V=800.0 PL=0
MOVL C01722 V=800.0 PL=0
MOVL C01723 V=800.0 PL=0
MOVL C01724 V=800.0 PL=0
MOVL C01725 V=800.0 PL=0
MOVL C01726 V=800.0 PL=0
MOVL C01727 V=800.0 PL=0
MOVL C01728 V=800.0 PL=0
MOVL C01729 V=800.0 PL=0
MOVL C01730 V=800.0 PL=0
MOVL C01731 V=800.0 PL=0
MOVL C01732 V=800.0 PL=0
MOVL C01733 V=800.0 PL=0
MOVL C01734 V=800.0 PL=0
MOVL C01735 V=800.0 PL=0
MOVL C01736 V=800.0 PL=0
MOVL C01737 V=800.0 PL=0
MOVL C01738 V=800.0 PL=0
MOVL C01739 V=800.0 PL=0
MOVL C01740 V=800.0 PL=0
MOVL C01741 V=800.0 PL=0
MOVL C01742 V=800.0 PL=0
MOVL C01743 V=800.0 PL=0
MOVL C01744 V=800.0 PL=0
MOVL C01745 V=800.0 PL=0
MOVL C01746 V=800.0 PL=0
MOVL C01747 V=800.0 PL=0
MOVL C01748 V=800.0 PL=0
MOVL C01749 V=800.0 PL=0
MOVL C01750 V=800.0 PL=0
MOVL C01751 V=800.0 PL=0
MOVL C01752 V=800.0 PL=0
MOVL C01753 V=800.0 PL=0
MOVL C01754 V=800.0 PL=0
MOVL C01755 V=800.0 PL=0
MOVL C01756 V=800.0 PL=0
MOVL C01757 V=800.0 PL=0
MOVL C01758 V=800.0 PL=0
MOVL C01759 V=800.0 PL=0
MOVL C01760 V=800.0 PL=0
MOVL C01761 V=800.0 PL=0
MOVL C01762 V=800.0 PL=0
MOVL C01763 V=800.0 PL=0
MOVL C01764 V=800.0 PL=0
MOVL C01765 V=800.0 PL=0
MOVL C01766 V=800.0 PL=0
MOVL C01767 V=800.0 PL=0
MOVL C01768 V=800.0 PL=0
MOVL C01769 V=800.0 PL=0
MOVL C01770 V=800.0 PL=0
MOVL C01771 V=800.0 PL=0
MOVL C01772 V=800.0 PL=0
MOVL C01773 V=800.0 PL=0
MOVL C01774 V=800.0 PL=0
MOVL C01775 V=800.0 PL=0
MOVL C01776 V=800.0 PL=0
MOVL C01777 V=800.0 PL=0
MOVL C01778 V=800.0 PL=0
MOVL C01779 V=800.0 PL=0
MOVL C01780 V=800.0 PL=0
MOVL C01781 V=800.0 PL=0
MOVL C01782 V=800.0 PL=0
MOVL C01783 V=800.0 PL=0
MOVL C01784 V=800.0 PL=0
MOVL C01785 V=800.0 PL=0
MOVL C01786 V=800.0 PL=0
MOVL C01787 V=800.0 PL=0
MOVL C01788 V=800.0 PL=0
MOVL C01789 V=800.0 PL=0
MOVL C01790 V=800.0 PL=0
MOVL C01791 V=800.0 PL=0
MOVL C01792 V=800.0 PL=0
MOVL C01793 V=800.0 PL=0
MOVL C01794 V=800.0 PL=0
MOVL C01795 V=800.0 PL=0
MOVL C01796 V=800.0 PL=0
MOVL C01797 V=800.0 PL=0
MOVL C01798 V=800.0 PL=0
MOVL C01799 V=800.0 PL=0
MOVL C01800 V=800.0 PL=0
MOVL C01801 V=800.0 PL=0
MOVL C01802 V=800.0 PL=0
MOVL C01803 V=800.0 PL=0
MOVL C01804 V=800.0 PL=0
MOVL C01805 V=800.0 PL=0
MOVL C01806 V=800.0 PL=0
MOVL C01807 V=800.0 PL=0
MOVL C01808 V=800.0 PL=0
MOVL C01809 V=800.0 PL=0
MOVL C01810 V=800.0 PL=0
MOVL C01811 V=800.0 PL=0
MOVL C01812 V=800.0 PL=0
MOVL C01813 V=800.0 PL=0
MOVL C01814 V=800.0 PL=0
MOVL C01815 V=800.0 PL=0
MOVL C01816 V=800.0 PL=0
MOVL C01817 V=800.0 PL=0
MOVL C01818 V=800.0 PL=0
MOVL C01819 V=800.0 PL=0
MOVL C01820 V=800.0 PL=0
MOVL C01821 V=800.0 PL=0
MOVL C01822 V=800.0 PL=0
MOVL C01823 V=800.0 PL=0
MOVL C01824 V=800.0 PL=0
MOVL C01825 V=800.0 PL=0
MOVL C01826 V=800.0 PL=0
MOVL C01827 V=800.0 PL=0
MOVL C01828 V=800.0 PL=0
MOVL C01829 V=800.0 PL=0
MOVL C01830 V=800.0 PL=0
MOVL C01831 V=800.0 PL=0
MOVL C01832 V=800.0 PL=0
MOVL C01833 V=800.0 PL=0
MOVL C01834 V=800.0 PL=0
MOVL C01835 V=800.0 PL=0
MOVL C01836 V=800.0 PL=0
MOVL C01837 V=800.0 PL=0
MOVL C01838 V=800.0 PL=0
MOVL C01839 V=800.0 PL=0
MOVL C01840 V=800.0 PL=0
MOVL C01841 V=800.0 PL=0
MOVL C01842 V=800.0 PL=0
MOVL C01843 V=800.0 PL=0
MOVL C01844 V=800.0 PL=0
MOVL C01845 V=800.0 PL=0
MOVL C01846 V=800.0 PL=0
MOVL C01847 V=800.0 PL=0
MOVL C01848 V=800.0 PL=0
MOVL C01849 V=800.0 PL=0
MOVL C01850 V=800.0 PL=0
MOVL C01851 V=800.0 PL=0
MOVL C01852 V=800.0 PL=0
MOVL C01853 V=800.0 PL=0
MOVL C01854 V=800.0 PL=0
MOVL C01855 V=800.0 PL=0
MOVL C01856 V=800.0 PL=0
MOVL C01857 V=800.0 PL=0
MOVL C01858 V=800.0 PL=0
MOVL C01859 V=800.0 PL=0
MOVL C01860 V=800.0 PL=0
MOVL C01861 V=800.0 PL=0
MOVL C01862 V=800.0 PL=0
MOVL C01863 V=800.0 PL=0
MOVL C01864 V=800.0 PL=0
MOVL C01865 V=800.0 PL=0
MOVL C01866 V=800.0 PL=0
MOVL C01867 V=800.0 PL=0
MOVL C01868 V=800.0 PL=0
MOVL C01869 V=800.0 PL=0
MOVL C01870 V=800.0 PL=0
MOVL C01871 V=800.0 PL=0
MOVL C01872 V=800.0 PL=0
MOVL C01873 V=800.0 PL=0
MOVL C01874 V=800.0 PL=0
MOVL C01875 V=800.0 PL=0
MOVL C01876 V=800.0 PL=0
MOVL C01877 V=800.0 PL=0
MOVL C01878 V=800.0 PL=0
MOVL C01879 V=800.0 PL=0
MOVL C01880 V=800.0 PL=0
MOVL C01881 V=800.0 PL=0
MOVL C01882 V=800.0 PL=0
MOVL C01883 V=800.0 PL=0
MOVL C01884 V=800.0 PL=0
MOVL C01885 V=800.0 PL=0
MOVL C01886 V=800.0 PL=0
MOVL C01887 V=800.0 PL=0
MOVL C01888 V=800.0 PL=0
MOVL C01889 V=800.0 PL=0
MOVL C01890 V=800.0 PL=0
MOVL C01891 V=800.0 PL=0
MOVL C01892 V=800.0 PL=0
MOVL C01893 V=800.0 PL=0
MOVL C01894 V=800.0 PL=0
MOVL C01895 V=800.0 PL=0
MOVL C01896 V=800.0 PL=0
MOVL C01897 V=800.0 PL=0
MOVL C01898 V=800.0 PL=0
MOVL C01899 V=800.0 PL=0
MOVL C01900 V=800.0 PL=0
MOVL C01901 V=800.0 PL=0
MOVL C01902 V=800.0 PL=0
MOVL C01903 V=800.0 PL=0
MOVL C01904 V=800.0 PL=0
MOVL C01905 V=800.0 PL=0
MOVL C01906 V=800.0 PL=0
MOVL C01907 V=800.0 PL=0
MOVL C01908 V=800.0 PL=0
MOVL C01909 V=800.0 PL=0
MOVL C01910 V=800.0 PL=0
MOVL C01911 V=800.0 PL=0
MOVL C01912 V=800.0 PL=0
MOVL C01913 V=800.0 PL=0
MOVL C01914 V=800.0 PL=0
MOVL C01915 V=800.0 PL=0
MOVL C01916 V=800.0 PL=0
MOVL C01917 V=800.0 PL=0
MOVL C01918 V=800.0 PL=0
MOVL C01919 V=800.0 PL=0
MOVL C01920 V=800.0 PL=0
MOVL C01921 V=800.0 PL=0
MOVL C01922 V=800.0 PL=0
MOVL C01923 V=800.0 PL=0
MOVL C01924 V=800.0 PL=0
MOVL C01925 V=800.0 PL=0
MOVL C01926 V=800.0 PL=0
MOVL C01927 V=800.0 PL=0
MOVL C01928 V=800.0 PL=0
MOVL C01929 V=800.0 PL=0
MOVL C01930 V=800.0 PL=0
MOVL C01931 V=800.0 PL=0
MOVL C01932 V=800.0 PL=0
MOVL C01933 V=800.0 PL=0
MOVL C01934 V=800.0 PL=0
MOVL C01935 V=800.0 PL=0
MOVL C01936 V=800.0 PL=0
MOVL C01937 V=800.0 PL=0
MOVL C01938 V=800.0 PL=0
MOVL C01939 V=800.0 PL=0
MOVL C01940 V=800.0 PL=0
MOVL C01941 V=800.0 PL=0
MOVL C01942 V=800.0 PL=0
MOVL C01943 V=800.0 PL=0
MOVL C01944 V=800.0 PL=0
MOVL C01945 V=800.0 PL=0
MOVL C01946 V=800.0 PL=0
MOVL C01947 V=800.0 PL=0
MOVL C01948 V=800.0 PL=0
MOVL C01949 V=800.0 PL=0
MOVL C01950 V=800.0 PL=0
MOVL C01951 V=800.0 PL=0
MOVL C01952 V=800.0 PL=0
MOVL C01953 V=800.0 PL=0
MOVL C01954 V=800.0 PL=0
MOVL C01955 V=800.0 PL=0
MOVL C01956 V=800.0 PL=0
MOVL C01957 V=800.0 PL=0
MOVL C01958 V=800.0 PL=0
MOVL C01959 V=800.0 PL=0
MOVL C01960 V=800.0 PL=0
MOVL C01961 V=800.0 PL=0
MOVL C01962 V=800.0 PL=0
MOVL C01963 V=800.0 PL=0
MOVL C01964 V=800.0 PL=0
MOVL C01965 V=800.0 PL=0
MOVL C01966 V=800.0 PL=0
MOVL C01967 V=800.0 PL=0
MOVL C01968 V=800.0 PL=0
MOVL C01969 V=800.0 PL=0
MOVL C01970 V=800.0 PL=0
MOVL C01971 V=800.0 PL=0
MOVL C01972 V=800.0 PL=0
MOVL C01973 V=800.0 PL=0
MOVL C01974 V=800.0 PL=0
MOVL C01975 V=800.0 PL=0
MOVL C01976 V=800.0 PL=0
MOVL C01977 V=800.0 PL=0
MOVL C01978 V=800.0 PL=0
MOVL C01979 V=800.0 PL=0
MOVL C01980 V=800.0 PL=0
MOVL C01981 V=800.0 PL=0
MOVL C01982 V=800.0 PL=0
MOVL C01983 V=800.0 PL=0
MOVL C01984 V=800.0 PL=0
MOVL C01985 V=800.0 PL=0
MOVL C01986 V=800.0 PL=0
MOVL C01987 V=800.0 PL=0
MOVL C01988 V=800.0 PL=0
MOVL C01989 V=800.0 PL=0
MOVL C01990 V=800.0 PL=0
MOVL C01991 V=800.0 PL=0
MOVL C01992 V=800.0 PL=0
MOVL C01993 V=800.0 PL=0
MOVL C01994 V=800.0 PL=0
MOVL C01995 V=800.0 PL=0
MOVL C01996 V=800.0 PL=0
MOVL C01997 V=800.0 PL=0
MOVL C01998 V=800.0 PL=0
MOVL C01999 V=800.0 PL=0
MOVL C02000 V=800.0 PL=0
MOVL C02001 V=800.0 PL=0
MOVL C02002 V=800.0 PL=0
MOVL C02003 V=800.0 PL=0
